KUKA KRL program: f1_Kuka_APT217T03S17.SRC

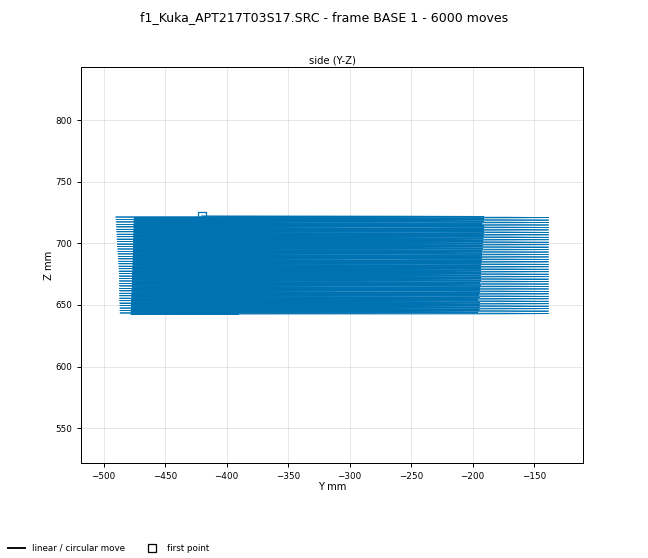
[picture p0: tool path of f1_Kuka_APT217T03S17.SRC in frame BASE 1, 6000 of 6001 moves have a stored position in this frame; points joined in program order, loops and branches not executed]
&ACCESS RVP
&REL 2
&PARAM TEMPLATE = C:\KRC\Roboter\Template\vorgabe
&PARAM EDITMASK = *
DEF f1_Kuka_APT217T03S17()


;FOLD INI;%{PE}%V3.2.0,%MKUKATPBASIS,%CINIT,%VCOMMON,%P
  ;FOLD BAS INI;%{E}%V3.2.0,%MKUKATPBASIS,%CINIT,%VINIT,%P
    GLOBAL INTERRUPT DECL 3 WHEN $STOPMESS==TRUE DO IR_STOPM ( )
    INTERRUPT ON 3
    BAS (#INITMOV,0 )
  ;ENDFOLD (BAS INI)
  ;FOLD USER INI;%{E}%V3.2.0,%MKUKATPUSER,%CINIT,%VINIT,%P
    ;Make your modifications here
  ;ENDFOLD (USER INI)
;ENDFOLD (INI)


;*** Make Null PTP Move
  PTP $pos_act

;*** Auto Load The Correct TOOL Data
  $tool=tool_data[3]

;*** Auto Load The Correct BASE Data
  $base=base_data[1]

  $ADVANCE = 5

;*** Restate Last Velocity
MMPM(30000.0)
SetRPM(6000)
LIN {X -0.045,Y -420.366,Z 722.490,A 0.000,B 0.000,C 90.000,E1 88.282} C_DIS
LIN {X -0.153,Y -409.375,Z 722.480,A 0.000,B 0.000,C 90.000,E1 86.388} C_DIS
LIN {X -0.011,Y -396.739,Z 722.467,A 0.000,B 0.000,C 90.000,E1 84.147} C_DIS
LIN {X -0.054,Y -382.651,Z 722.453,A 0.000,B 0.000,C 90.000,E1 81.602} C_DIS
LIN {X -0.034,Y -370.606,Z 722.440,A 0.000,B 0.000,C 90.000,E1 79.285} C_DIS
LIN {X -0.131,Y -357.568,Z 722.426,A 0.000,B 0.000,C 90.000,E1 76.645} C_DIS
LIN {X 0.016,Y -346.347,Z 722.412,A 0.000,B 0.000,C 90.000,E1 74.212} C_DIS
LIN {X -0.021,Y -335.329,Z 722.399,A 0.000,B 0.000,C 90.000,E1 71.764} C_DIS
LIN {X 0.156,Y -320.932,Z 722.380,A 0.000,B 0.000,C 90.000,E1 68.284} C_DIS
LIN {X 0.051,Y -311.481,Z 722.365,A 0.000,B 0.000,C 90.000,E1 65.741} C_DIS
LIN {X 0.067,Y -300.034,Z 722.345,A 0.000,B 0.000,C 90.000,E1 62.153} C_DIS
LIN {X -0.118,Y -290.423,Z 722.327,A 0.000,B 0.000,C 90.000,E1 58.869} C_DIS
LIN {X -0.001,Y -281.361,Z 722.308,A 0.000,B 0.000,C 90.000,E1 55.468} C_DIS
LIN {X -0.016,Y -276.153,Z 722.297,A 0.000,B 0.000,C 90.000,E1 53.417} C_DIS
LIN {X 0.036,Y -270.874,Z 722.285,A 0.000,B 0.000,C 90.000,E1 51.331} C_DIS
LIN {X 0.116,Y -265.448,Z 722.274,A 0.000,B 0.000,C 90.000,E1 49.218} C_DIS
LIN {X -0.099,Y -259.838,Z 722.262,A 0.000,B 0.000,C 90.000,E1 47.148} C_DIS
LIN {X -0.064,Y -254.168,Z 722.250,A 0.000,B 0.000,C 90.000,E1 45.000} C_DIS
LIN {X -0.132,Y -248.317,Z 722.238,A 0.000,B 0.000,C 90.000,E1 42.852} C_DIS
LIN {X 0.051,Y -242.351,Z 722.226,A 0.000,B 0.000,C 90.000,E1 40.620} C_DIS
LIN {X -0.106,Y -232.554,Z 722.205,A 0.000,B 0.000,C 90.000,E1 36.950} C_DIS
LIN {X -0.091,Y -223.507,Z 722.184,A 0.000,B 0.000,C 90.000,E1 33.166} C_DIS
LIN {X -0.050,Y -216.883,Z 722.167,A 0.000,B 0.000,C 90.000,E1 30.079} C_DIS
LIN {X -0.011,Y -211.033,Z 722.150,A 0.000,B 0.000,C 90.000,E1 26.950} C_DIS
LIN {X 0.066,Y -205.943,Z 722.132,A 0.000,B 0.000,C 90.000,E1 23.770} C_DIS
LIN {X -0.046,Y -201.601,Z 722.114,A 0.000,B 0.000,C 90.000,E1 20.610} C_DIS
LIN {X -0.008,Y -197.203,Z 722.092,A 0.000,B 0.000,C 90.000,E1 16.567} C_DIS
LIN {X 0.070,Y -193.392,Z 722.065,A 0.000,B 0.000,C 90.000,E1 11.658} C_DIS
LIN {X 0.073,Y -190.840,Z 722.033,A 0.000,B 0.000,C 90.000,E1 5.910} C_DIS
LIN {X -0.076,Y -191.951,Z 721.970,A 0.000,B 0.000,C 90.000,E1 354.609} C_DIS
LIN {X -0.101,Y -194.807,Z 721.943,A 0.000,B 0.000,C 90.000,E1 349.690} C_DIS
LIN {X -0.024,Y -198.321,Z 721.920,A 0.000,B 0.000,C 90.000,E1 345.589} C_DIS
LIN {X 0.030,Y -202.840,Z 721.897,A 0.000,B 0.000,C 90.000,E1 341.529} C_DIS
LIN {X -0.017,Y -208.249,Z 721.875,A 0.000,B 0.000,C 90.000,E1 337.539} C_DIS
LIN {X -0.036,Y -214.509,Z 721.853,A 0.000,B 0.000,C 90.000,E1 333.589} C_DIS
LIN {X 0.047,Y -221.349,Z 721.832,A 0.000,B 0.000,C 90.000,E1 329.665} C_DIS
LIN {X 0.069,Y -227.297,Z 721.814,A 0.000,B 0.000,C 90.000,E1 326.580} C_DIS
LIN {X 0.013,Y -235.274,Z 721.793,A 0.000,B 0.000,C 90.000,E1 322.798} C_DIS
LIN {X 0.048,Y -243.974,Z 721.773,A 0.000,B 0.000,C 90.000,E1 319.057} C_DIS
LIN {X -0.019,Y -253.622,Z 721.752,A 0.000,B 0.000,C 90.000,E1 315.405} C_DIS
LIN {X -0.120,Y -264.412,Z 721.732,A 0.000,B 0.000,C 90.000,E1 311.838} C_DIS
LIN {X -0.010,Y -276.297,Z 721.713,A 0.000,B 0.000,C 90.000,E1 308.302} C_DIS
LIN {X -0.150,Y -289.563,Z 721.694,A 0.000,B 0.000,C 90.000,E1 304.898} C_DIS
LIN {X -0.111,Y -304.342,Z 721.675,A 0.000,B 0.000,C 90.000,E1 301.544} C_DIS
LIN {X -0.142,Y -319.094,Z 721.659,A 0.000,B 0.000,C 90.000,E1 298.615} C_DIS
LIN {X 0.051,Y -337.144,Z 721.641,A 0.000,B 0.000,C 90.000,E1 295.412} C_DIS
LIN {X 0.060,Y -354.682,Z 721.626,A 0.000,B 0.000,C 90.000,E1 292.642} C_DIS
LIN {X -0.097,Y -375.452,Z 721.609,A 0.000,B 0.000,C 90.000,E1 289.685} C_DIS
LIN {X -0.149,Y -396.197,Z 721.595,A 0.000,B 0.000,C 90.000,E1 287.094} C_DIS
LIN {X 0.119,Y -410.310,Z 721.586,A 0.000,B 0.000,C 90.000,E1 285.371} C_DIS
LIN {X 0.155,Y -424.096,Z 721.576,A 0.000,B 0.000,C 90.000,E1 283.716} C_DIS
LIN {X -0.176,Y -435.418,Z 721.569,A 0.000,B 0.000,C 90.000,E1 282.411} C_DIS
LIN {X 0.197,Y -444.037,Z 721.563,A 0.000,B 0.000,C 90.000,E1 281.299} C_DIS
LIN {X -0.035,Y -454.322,Z 721.556,A 0.000,B 0.000,C 90.000,E1 280.018} C_DIS
LIN {X 0.089,Y -466.419,Z 721.547,A 0.000,B 0.000,C 90.000,E1 278.454} C_DIS
LIN {X -0.153,Y -473.979,Z 721.541,A 0.000,B 0.000,C 90.000,E1 277.466} C_DIS
LIN {X -0.243,Y -478.914,Z 721.537,A 0.000,B 0.000,C 90.000,E1 276.720} C_DIS
LIN {X -0.096,Y -481.792,Z 721.534,A 0.000,B 0.000,C 90.000,E1 276.201} C_DIS
LIN {X 0.070,Y -484.223,Z 721.532,A 0.000,B 0.000,C 90.000,E1 275.682} C_DIS
LIN {X -0.232,Y -486.263,Z 721.529,A 0.000,B 0.000,C 90.000,E1 275.220} C_DIS
LIN {X -0.045,Y -487.865,Z 721.526,A 0.000,B 0.000,C 90.000,E1 274.702} C_DIS
LIN {X 0.115,Y -489.063,Z 721.523,A 0.000,B 0.000,C 90.000,E1 274.188} C_DIS
LIN {X -0.166,Y -489.824,Z 721.521,A 0.000,B 0.000,C 90.000,E1 273.726} C_DIS
LIN {X 0.017,Y -490.215,Z 721.518,A 0.000,B 0.000,C 90.000,E1 273.212} C_DIS
LIN {X 0.233,Y -490.237,Z 721.515,A 0.000,B 0.000,C 90.000,E1 272.694} C_DIS
LIN {X -0.063,Y -489.908,Z 721.512,A 0.000,B 0.000,C 90.000,E1 272.236} C_DIS
LIN {X 0.148,Y -489.291,Z 721.510,A 0.000,B 0.000,C 90.000,E1 271.718} C_DIS
LIN {X -0.148,Y -488.268,Z 721.507,A 0.000,B 0.000,C 90.000,E1 271.260} C_DIS
LIN {X 0.041,Y -486.857,Z 721.504,A 0.000,B 0.000,C 90.000,E1 270.745} C_DIS
LIN {X 0.225,Y -484.965,Z 721.501,A 0.000,B 0.000,C 90.000,E1 270.229} C_DIS
LIN {X -0.083,Y -482.513,Z 721.499,A 0.000,B 0.000,C 90.000,E1 269.771} C_DIS
LIN {X 0.074,Y -479.349,Z 721.496,A 0.000,B 0.000,C 90.000,E1 269.255} C_DIS
LIN {X 0.212,Y -475.359,Z 721.493,A 0.000,B 0.000,C 90.000,E1 268.740} C_DIS
LIN {X -0.144,Y -470.353,Z 721.490,A 0.000,B 0.000,C 90.000,E1 268.282} C_DIS
LIN {X -0.225,Y -467.502,Z 721.489,A 0.000,B 0.000,C 90.000,E1 268.051} C_DIS
LIN {X 0.144,Y -464.309,Z 721.488,A 0.000,B 0.000,C 90.000,E1 267.764} C_DIS
LIN {X 0.057,Y -457.761,Z 721.485,A 0.000,B 0.000,C 90.000,E1 267.364} C_DIS
LIN {X 0.057,Y -454.413,Z 721.484,A 0.000,B 0.000,C 90.000,E1 267.192} C_DIS
LIN {X -0.086,Y -447.138,Z 721.483,A 0.000,B 0.000,C 90.000,E1 266.906} C_DIS
LIN {X -0.114,Y -439.506,Z 721.481,A 0.000,B 0.000,C 90.000,E1 266.674} C_DIS
LIN {X -0.117,Y -431.202,Z 721.480,A 0.000,B 0.000,C 90.000,E1 266.502} C_DIS
LIN {X -0.201,Y -425.998,Z 721.480,A 0.000,B 0.000,C 90.000,E1 266.445} C_DIS
LIN {X -0.115,Y -419.753,Z 721.480,A 0.000,B 0.000,C 90.000,E1 266.388} C_DIS
LIN {X -0.086,Y -180.939,Z 721.480,A 0.000,B 0.000,C 90.000,E1 266.388} C_DIS
LIN {X -0.079,Y -180.742,Z 721.470,A 0.000,B 0.000,C 90.000,E1 264.666} C_DIS
LIN {X 0.022,Y -178.834,Z 721.442,A 0.000,B 0.000,C 90.000,E1 259.567} C_DIS
LIN {X 0.056,Y -175.878,Z 721.414,A 0.000,B 0.000,C 90.000,E1 254.464} C_DIS
LIN {X -0.007,Y -174.538,Z 721.404,A 0.000,B 0.000,C 90.000,E1 252.779} C_DIS
LIN {X 0.086,Y -171.522,Z 721.380,A 0.000,B 0.000,C 90.000,E1 248.465} C_DIS
LIN {X 0.071,Y -167.748,Z 721.357,A 0.000,B 0.000,C 90.000,E1 244.152} C_DIS
LIN {X 0.010,Y -166.451,Z 721.347,A 0.000,B 0.000,C 90.000,E1 242.436} C_DIS
LIN {X 0.000,Y -163.167,Z 721.328,A 0.000,B 0.000,C 90.000,E1 238.948} C_DIS
LIN {X 0.049,Y -161.126,Z 721.313,A 0.000,B 0.000,C 90.000,E1 236.294} C_DIS
LIN {X -0.048,Y -157.149,Z 721.288,A 0.000,B 0.000,C 90.000,E1 231.904} C_DIS
LIN {X -0.025,Y -155.880,Z 721.278,A 0.000,B 0.000,C 90.000,E1 230.114} C_DIS
LIN {X -0.066,Y -152.131,Z 721.253,A 0.000,B 0.000,C 90.000,E1 225.648} C_DIS
LIN {X -0.046,Y -150.381,Z 721.238,A 0.000,B 0.000,C 90.000,E1 222.933} C_DIS
LIN {X -0.021,Y -147.113,Z 721.213,A 0.000,B 0.000,C 90.000,E1 218.382} C_DIS
LIN {X -0.030,Y -145.679,Z 721.198,A 0.000,B 0.000,C 90.000,E1 215.644} C_DIS
LIN {X -0.032,Y -143.061,Z 721.172,A 0.000,B 0.000,C 90.000,E1 211.052} C_DIS
LIN {X 0.025,Y -141.683,Z 721.152,A 0.000,B 0.000,C 90.000,E1 207.334} C_DIS
LIN {X 0.004,Y -139.458,Z 721.116,A 0.000,B 0.000,C 90.000,E1 200.844} C_DIS
LIN {X 0.055,Y -139.192,Z 721.105,A 0.000,B 0.000,C 90.000,E1 198.960} C_DIS
LIN {X -0.058,Y -138.324,Z 721.054,A 0.000,B 0.000,C 90.000,E1 189.670} C_DIS
LIN {X -0.054,Y -139.455,Z 721.007,A 0.000,B 0.000,C 90.000,E1 181.260} C_DIS
LIN {X 0.026,Y -141.003,Z 720.976,A 0.000,B 0.000,C 90.000,E1 175.641} C_DIS
LIN {X -0.024,Y -142.757,Z 720.955,A 0.000,B 0.000,C 90.000,E1 171.951} C_DIS
LIN {X -0.069,Y -145.160,Z 720.930,A 0.000,B 0.000,C 90.000,E1 167.353} C_DIS
LIN {X -0.077,Y -147.783,Z 720.909,A 0.000,B 0.000,C 90.000,E1 163.685} C_DIS
LIN {X 0.003,Y -150.462,Z 720.889,A 0.000,B 0.000,C 90.000,E1 160.007} C_DIS
LIN {X 0.077,Y -153.913,Z 720.869,A 0.000,B 0.000,C 90.000,E1 156.357} C_DIS
LIN {X 0.002,Y -157.323,Z 720.849,A 0.000,B 0.000,C 90.000,E1 152.794} C_DIS
LIN {X 0.086,Y -161.512,Z 720.829,A 0.000,B 0.000,C 90.000,E1 149.203} C_DIS
LIN {X -0.037,Y -165.711,Z 720.810,A 0.000,B 0.000,C 90.000,E1 145.722} C_DIS
LIN {X 0.088,Y -170.657,Z 720.790,A 0.000,B 0.000,C 90.000,E1 142.190} C_DIS
LIN {X 0.001,Y -175.533,Z 720.771,A 0.000,B 0.000,C 90.000,E1 138.771} C_DIS
LIN {X -0.006,Y -181.152,Z 720.752,A 0.000,B 0.000,C 90.000,E1 135.364} C_DIS
LIN {X -0.007,Y -186.606,Z 720.733,A 0.000,B 0.000,C 90.000,E1 132.000} C_DIS
LIN {X 0.028,Y -191.565,Z 720.718,A 0.000,B 0.000,C 90.000,E1 129.277} C_DIS
LIN {X 0.008,Y -290.263,Z 720.718,A 0.000,B 0.000,C 90.000,E1 129.277} C_DIS
LIN {X 0.150,Y -292.744,Z 720.718,A 0.000,B 0.000,C 90.000,E1 129.197} C_DIS
LIN {X -0.022,Y -297.486,Z 720.716,A 0.000,B 0.000,C 90.000,E1 128.955} C_DIS
LIN {X 0.033,Y -300.182,Z 720.715,A 0.000,B 0.000,C 90.000,E1 128.669} C_DIS
LIN {X 0.012,Y -303.878,Z 720.712,A 0.000,B 0.000,C 90.000,E1 128.096} C_DIS
LIN {X 0.204,Y -305.355,Z 720.710,A 0.000,B 0.000,C 90.000,E1 127.729} C_DIS
LIN {X -0.032,Y -306.516,Z 720.708,A 0.000,B 0.000,C 90.000,E1 127.443} C_DIS
LIN {X -0.049,Y -317.229,Z 720.688,A 0.000,B 0.000,C 90.000,E1 123.865} C_DIS
LIN {X -0.123,Y -327.331,Z 720.672,A 0.000,B 0.000,C 90.000,E1 121.003} C_DIS
LIN {X 0.034,Y -338.764,Z 720.656,A 0.000,B 0.000,C 90.000,E1 118.153} C_DIS
LIN {X -0.121,Y -351.632,Z 720.641,A 0.000,B 0.000,C 90.000,E1 115.412} C_DIS
LIN {X 0.208,Y -364.364,Z 720.628,A 0.000,B 0.000,C 90.000,E1 112.950} C_DIS
LIN {X 0.099,Y -378.411,Z 720.615,A 0.000,B 0.000,C 90.000,E1 110.610} C_DIS
LIN {X 0.079,Y -393.872,Z 720.602,A 0.000,B 0.000,C 90.000,E1 108.308} C_DIS
LIN {X -0.062,Y -410.861,Z 720.589,A 0.000,B 0.000,C 90.000,E1 106.079} C_DIS
LIN {X -0.026,Y -429.500,Z 720.577,A 0.000,B 0.000,C 90.000,E1 103.883} C_DIS
LIN {X 0.195,Y -449.465,Z 720.566,A 0.000,B 0.000,C 90.000,E1 101.771} C_DIS
LIN {X -0.208,Y -467.386,Z 720.556,A 0.000,B 0.000,C 90.000,E1 100.141} C_DIS
LIN {X -0.172,Y -469.669,Z 720.555,A 0.000,B 0.000,C 90.000,E1 99.905} C_DIS
LIN {X 0.177,Y -471.507,Z 720.554,A 0.000,B 0.000,C 90.000,E1 99.613} C_DIS
LIN {X 0.061,Y -472.893,Z 720.552,A 0.000,B 0.000,C 90.000,E1 99.378} C_DIS
LIN {X 0.168,Y -474.683,Z 720.549,A 0.000,B 0.000,C 90.000,E1 98.859} C_DIS
LIN {X -0.185,Y -475.386,Z 720.547,A 0.000,B 0.000,C 90.000,E1 98.398} C_DIS
LIN {X 0.010,Y -475.120,Z 720.544,A 0.000,B 0.000,C 90.000,E1 97.871} C_DIS
LIN {X 0.142,Y -473.850,Z 720.541,A 0.000,B 0.000,C 90.000,E1 97.352} C_DIS
LIN {X -0.056,Y -472.778,Z 720.540,A 0.000,B 0.000,C 90.000,E1 97.125} C_DIS
LIN {X 0.071,Y -469.662,Z 720.537,A 0.000,B 0.000,C 90.000,E1 96.606} C_DIS
LIN {X -0.074,Y -453.400,Z 720.523,A 0.000,B 0.000,C 90.000,E1 94.073} C_DIS
LIN {X 0.011,Y -440.049,Z 720.510,A 0.000,B 0.000,C 90.000,E1 91.718} C_DIS
LIN {X 0.130,Y -431.084,Z 720.501,A 0.000,B 0.000,C 90.000,E1 90.115} C_DIS
LIN {X -0.215,Y -420.296,Z 720.490,A 0.000,B 0.000,C 90.000,E1 88.282} C_DIS
LIN {X 0.088,Y -409.303,Z 720.480,A 0.000,B 0.000,C 90.000,E1 86.331} C_DIS
LIN {X -0.174,Y -396.689,Z 720.467,A 0.000,B 0.000,C 90.000,E1 84.147} C_DIS
LIN {X 0.200,Y -381.112,Z 720.452,A 0.000,B 0.000,C 90.000,E1 81.254} C_DIS
LIN {X -0.189,Y -369.132,Z 720.439,A 0.000,B 0.000,C 90.000,E1 78.993} C_DIS
LIN {X 0.022,Y -356.168,Z 720.424,A 0.000,B 0.000,C 90.000,E1 76.297} C_DIS
LIN {X 0.123,Y -344.996,Z 720.410,A 0.000,B 0.000,C 90.000,E1 73.866} C_DIS
LIN {X 0.131,Y -332.686,Z 720.395,A 0.000,B 0.000,C 90.000,E1 71.094} C_DIS
LIN {X -0.081,Y -318.566,Z 720.376,A 0.000,B 0.000,C 90.000,E1 67.667} C_DIS
LIN {X -0.023,Y -310.507,Z 720.363,A 0.000,B 0.000,C 90.000,E1 65.409} C_DIS
LIN {X -0.049,Y -300.214,Z 720.345,A 0.000,B 0.000,C 90.000,E1 62.153} C_DIS
LIN {X 0.024,Y -290.640,Z 720.327,A 0.000,B 0.000,C 90.000,E1 58.820} C_DIS
LIN {X -0.097,Y -281.608,Z 720.308,A 0.000,B 0.000,C 90.000,E1 55.468} C_DIS
LIN {X -0.106,Y -276.420,Z 720.297,A 0.000,B 0.000,C 90.000,E1 53.417} C_DIS
LIN {X -0.048,Y -271.151,Z 720.285,A 0.000,B 0.000,C 90.000,E1 51.331} C_DIS
LIN {X 0.040,Y -265.742,Z 720.273,A 0.000,B 0.000,C 90.000,E1 49.218} C_DIS
LIN {X 0.022,Y -260.146,Z 720.262,A 0.000,B 0.000,C 90.000,E1 47.106} C_DIS
LIN {X -0.125,Y -254.445,Z 720.250,A 0.000,B 0.000,C 90.000,E1 45.000} C_DIS
LIN {X -0.018,Y -248.610,Z 720.238,A 0.000,B 0.000,C 90.000,E1 42.813} C_DIS
LIN {X 0.002,Y -242.609,Z 720.226,A 0.000,B 0.000,C 90.000,E1 40.620} C_DIS
LIN {X -0.005,Y -232.771,Z 720.205,A 0.000,B 0.000,C 90.000,E1 36.916} C_DIS
LIN {X -0.122,Y -223.698,Z 720.184,A 0.000,B 0.000,C 90.000,E1 33.166} C_DIS
LIN {X 0.033,Y -217.037,Z 720.167,A 0.000,B 0.000,C 90.000,E1 30.050} C_DIS
LIN {X -0.032,Y -211.188,Z 720.150,A 0.000,B 0.000,C 90.000,E1 26.950} C_DIS
LIN {X 0.049,Y -206.089,Z 720.132,A 0.000,B 0.000,C 90.000,E1 23.770} C_DIS
LIN {X -0.060,Y -201.735,Z 720.114,A 0.000,B 0.000,C 90.000,E1 20.610} C_DIS
LIN {X 0.040,Y -197.327,Z 720.092,A 0.000,B 0.000,C 90.000,E1 16.551} C_DIS
LIN {X 0.054,Y -194.024,Z 720.069,A 0.000,B 0.000,C 90.000,E1 12.479} C_DIS
LIN {X -0.073,Y -191.194,Z 720.038,A 0.000,B 0.000,C 90.000,E1 6.777} C_DIS
LIN {X 0.076,Y -192.439,Z 719.965,A 0.000,B 0.000,C 90.000,E1 353.742} C_DIS
LIN {X -0.084,Y -195.552,Z 719.938,A 0.000,B 0.000,C 90.000,E1 348.870} C_DIS
LIN {X 0.067,Y -199.250,Z 719.915,A 0.000,B 0.000,C 90.000,E1 344.755} C_DIS
LIN {X 0.023,Y -203.948,Z 719.893,A 0.000,B 0.000,C 90.000,E1 340.732} C_DIS
LIN {X 0.013,Y -209.531,Z 719.871,A 0.000,B 0.000,C 90.000,E1 336.741} C_DIS
LIN {X 0.026,Y -215.881,Z 719.849,A 0.000,B 0.000,C 90.000,E1 332.794} C_DIS
LIN {X -0.028,Y -222.851,Z 719.827,A 0.000,B 0.000,C 90.000,E1 328.918} C_DIS
LIN {X -0.092,Y -230.456,Z 719.806,A 0.000,B 0.000,C 90.000,E1 325.102} C_DIS
LIN {X -0.097,Y -238.696,Z 719.785,A 0.000,B 0.000,C 90.000,E1 321.331} C_DIS
LIN {X 0.023,Y -247.740,Z 719.764,A 0.000,B 0.000,C 90.000,E1 317.595} C_DIS
LIN {X -0.121,Y -256.774,Z 719.746,A 0.000,B 0.000,C 90.000,E1 314.352} C_DIS
LIN {X -0.107,Y -267.869,Z 719.726,A 0.000,B 0.000,C 90.000,E1 310.782} C_DIS
LIN {X 0.056,Y -278.884,Z 719.709,A 0.000,B 0.000,C 90.000,E1 307.604} C_DIS
LIN {X 0.010,Y -292.442,Z 719.690,A 0.000,B 0.000,C 90.000,E1 304.199} C_DIS
LIN {X -0.039,Y -305.944,Z 719.673,A 0.000,B 0.000,C 90.000,E1 301.209} C_DIS
LIN {X -0.093,Y -319.107,Z 719.659,A 0.000,B 0.000,C 90.000,E1 298.615} C_DIS
LIN {X 0.103,Y -337.113,Z 719.641,A 0.000,B 0.000,C 90.000,E1 295.412} C_DIS
LIN {X 0.113,Y -354.597,Z 719.626,A 0.000,B 0.000,C 90.000,E1 292.642} C_DIS
LIN {X -0.043,Y -375.337,Z 719.609,A 0.000,B 0.000,C 90.000,E1 289.685} C_DIS
LIN {X -0.096,Y -396.044,Z 719.595,A 0.000,B 0.000,C 90.000,E1 287.094} C_DIS
LIN {X 0.171,Y -410.128,Z 719.586,A 0.000,B 0.000,C 90.000,E1 285.371} C_DIS
LIN {X -0.206,Y -423.888,Z 719.576,A 0.000,B 0.000,C 90.000,E1 283.772} C_DIS
LIN {X -0.127,Y -435.207,Z 719.569,A 0.000,B 0.000,C 90.000,E1 282.411} C_DIS
LIN {X 0.244,Y -443.843,Z 719.563,A 0.000,B 0.000,C 90.000,E1 281.299} C_DIS
LIN {X 0.010,Y -454.095,Z 719.556,A 0.000,B 0.000,C 90.000,E1 280.018} C_DIS
LIN {X 0.131,Y -466.190,Z 719.547,A 0.000,B 0.000,C 90.000,E1 278.454} C_DIS
LIN {X -0.113,Y -473.775,Z 719.541,A 0.000,B 0.000,C 90.000,E1 277.466} C_DIS
LIN {X -0.204,Y -478.702,Z 719.537,A 0.000,B 0.000,C 90.000,E1 276.720} C_DIS
LIN {X -0.058,Y -481.588,Z 719.534,A 0.000,B 0.000,C 90.000,E1 276.201} C_DIS
LIN {X 0.107,Y -484.034,Z 719.532,A 0.000,B 0.000,C 90.000,E1 275.682} C_DIS
LIN {X -0.196,Y -486.084,Z 719.529,A 0.000,B 0.000,C 90.000,E1 275.220} C_DIS
LIN {X -0.004,Y -487.694,Z 719.526,A 0.000,B 0.000,C 90.000,E1 274.702} C_DIS
LIN {X 0.156,Y -488.877,Z 719.523,A 0.000,B 0.000,C 90.000,E1 274.188} C_DIS
LIN {X -0.126,Y -489.635,Z 719.521,A 0.000,B 0.000,C 90.000,E1 273.726} C_DIS
LIN {X 0.056,Y -489.999,Z 719.518,A 0.000,B 0.000,C 90.000,E1 273.212} C_DIS
LIN {X -0.219,Y -490.051,Z 719.515,A 0.000,B 0.000,C 90.000,E1 272.751} C_DIS
LIN {X -0.027,Y -489.687,Z 719.512,A 0.000,B 0.000,C 90.000,E1 272.236} C_DIS
LIN {X 0.183,Y -489.091,Z 719.510,A 0.000,B 0.000,C 90.000,E1 271.718} C_DIS
LIN {X -0.115,Y -488.083,Z 719.507,A 0.000,B 0.000,C 90.000,E1 271.260} C_DIS
LIN {X 0.074,Y -486.677,Z 719.504,A 0.000,B 0.000,C 90.000,E1 270.745} C_DIS
LIN {X -0.228,Y -484.823,Z 719.501,A 0.000,B 0.000,C 90.000,E1 270.286} C_DIS
LIN {X -0.052,Y -482.380,Z 719.499,A 0.000,B 0.000,C 90.000,E1 269.771} C_DIS
LIN {X 0.103,Y -479.214,Z 719.496,A 0.000,B 0.000,C 90.000,E1 269.255} C_DIS
LIN {X -0.235,Y -475.261,Z 719.493,A 0.000,B 0.000,C 90.000,E1 268.797} C_DIS
LIN {X -0.116,Y -470.303,Z 719.490,A 0.000,B 0.000,C 90.000,E1 268.282} C_DIS
LIN {X -0.200,Y -467.490,Z 719.489,A 0.000,B 0.000,C 90.000,E1 268.051} C_DIS
LIN {X 0.167,Y -464.322,Z 719.488,A 0.000,B 0.000,C 90.000,E1 267.764} C_DIS
LIN {X -0.119,Y -461.259,Z 719.487,A 0.000,B 0.000,C 90.000,E1 267.593} C_DIS
LIN {X 0.057,Y -457.778,Z 719.485,A 0.000,B 0.000,C 90.000,E1 267.364} C_DIS
LIN {X 0.053,Y -450.582,Z 719.483,A 0.000,B 0.000,C 90.000,E1 267.020} C_DIS
LIN {X 0.210,Y -443.185,Z 719.482,A 0.000,B 0.000,C 90.000,E1 266.731} C_DIS
LIN {X -0.066,Y -435.015,Z 719.481,A 0.000,B 0.000,C 90.000,E1 266.560} C_DIS
LIN {X 0.107,Y -425.230,Z 719.480,A 0.000,B 0.000,C 90.000,E1 266.388} C_DIS
LIN {X 0.192,Y -417.389,Z 719.480,A 0.000,B 0.000,C 90.000,E1 266.331} C_DIS
LIN {X 0.048,Y -180.938,Z 719.480,A 0.000,B 0.000,C 90.000,E1 266.331} C_DIS
LIN {X 0.055,Y -180.736,Z 719.470,A 0.000,B 0.000,C 90.000,E1 264.609} C_DIS
LIN {X -0.024,Y -178.826,Z 719.442,A 0.000,B 0.000,C 90.000,E1 259.567} C_DIS
LIN {X 0.058,Y -175.870,Z 719.414,A 0.000,B 0.000,C 90.000,E1 254.448} C_DIS
LIN {X 0.052,Y -173.843,Z 719.399,A 0.000,B 0.000,C 90.000,E1 251.891} C_DIS
LIN {X 0.041,Y -171.511,Z 719.380,A 0.000,B 0.000,C 90.000,E1 248.465} C_DIS
LIN {X 0.028,Y -167.738,Z 719.356,A 0.000,B 0.000,C 90.000,E1 244.152} C_DIS
LIN {X 0.044,Y -166.437,Z 719.347,A 0.000,B 0.000,C 90.000,E1 242.410} C_DIS
LIN {X -0.043,Y -163.155,Z 719.327,A 0.000,B 0.000,C 90.000,E1 238.948} C_DIS
LIN {X 0.007,Y -161.112,Z 719.313,A 0.000,B 0.000,C 90.000,E1 236.294} C_DIS
LIN {X -0.010,Y -157.837,Z 719.293,A 0.000,B 0.000,C 90.000,E1 232.763} C_DIS
LIN {X 0.053,Y -155.870,Z 719.278,A 0.000,B 0.000,C 90.000,E1 230.070} C_DIS
LIN {X 0.001,Y -152.120,Z 719.253,A 0.000,B 0.000,C 90.000,E1 225.607} C_DIS
LIN {X 0.016,Y -150.370,Z 719.238,A 0.000,B 0.000,C 90.000,E1 222.894} C_DIS
LIN {X -0.062,Y -147.104,Z 719.213,A 0.000,B 0.000,C 90.000,E1 218.382} C_DIS
LIN {X 0.048,Y -145.673,Z 719.198,A 0.000,B 0.000,C 90.000,E1 215.598} C_DIS
LIN {X 0.051,Y -143.054,Z 719.172,A 0.000,B 0.000,C 90.000,E1 211.003} C_DIS
LIN {X -0.013,Y -141.677,Z 719.152,A 0.000,B 0.000,C 90.000,E1 207.334} C_DIS
LIN {X -0.035,Y -139.455,Z 719.116,A 0.000,B 0.000,C 90.000,E1 200.844} C_DIS
LIN {X 0.016,Y -139.189,Z 719.105,A 0.000,B 0.000,C 90.000,E1 198.960} C_DIS
LIN {X 0.039,Y -138.323,Z 719.053,A 0.000,B 0.000,C 90.000,E1 189.613} C_DIS
LIN {X 0.046,Y -139.458,Z 719.007,A 0.000,B 0.000,C 90.000,E1 181.203} C_DIS
LIN {X -0.013,Y -141.009,Z 718.976,A 0.000,B 0.000,C 90.000,E1 175.641} C_DIS
LIN {X -0.064,Y -142.763,Z 718.955,A 0.000,B 0.000,C 90.000,E1 171.951} C_DIS
LIN {X 0.033,Y -145.170,Z 718.930,A 0.000,B 0.000,C 90.000,E1 167.297} C_DIS
LIN {X 0.025,Y -147.792,Z 718.909,A 0.000,B 0.000,C 90.000,E1 163.630} C_DIS
LIN {X -0.039,Y -150.475,Z 718.889,A 0.000,B 0.000,C 90.000,E1 160.007} C_DIS
LIN {X 0.036,Y -153.929,Z 718.869,A 0.000,B 0.000,C 90.000,E1 156.357} C_DIS
LIN {X -0.041,Y -157.339,Z 718.849,A 0.000,B 0.000,C 90.000,E1 152.794} C_DIS
LIN {X 0.043,Y -161.532,Z 718.829,A 0.000,B 0.000,C 90.000,E1 149.203} C_DIS
LIN {X 0.056,Y -165.730,Z 718.809,A 0.000,B 0.000,C 90.000,E1 145.674} C_DIS
LIN {X 0.044,Y -170.680,Z 718.790,A 0.000,B 0.000,C 90.000,E1 142.190} C_DIS
LIN {X -0.043,Y -175.555,Z 718.771,A 0.000,B 0.000,C 90.000,E1 138.771} C_DIS
LIN {X 0.076,Y -181.173,Z 718.752,A 0.000,B 0.000,C 90.000,E1 135.324} C_DIS
LIN {X -0.054,Y -186.631,Z 718.733,A 0.000,B 0.000,C 90.000,E1 132.000} C_DIS
LIN {X 0.072,Y -191.544,Z 718.718,A 0.000,B 0.000,C 90.000,E1 129.277} C_DIS
LIN {X 0.058,Y -290.577,Z 718.718,A 0.000,B 0.000,C 90.000,E1 129.277} C_DIS
LIN {X 0.043,Y -295.194,Z 718.717,A 0.000,B 0.000,C 90.000,E1 129.116} C_DIS
LIN {X -0.109,Y -297.362,Z 718.716,A 0.000,B 0.000,C 90.000,E1 128.991} C_DIS
LIN {X -0.040,Y -300.349,Z 718.715,A 0.000,B 0.000,C 90.000,E1 128.669} C_DIS
LIN {X -0.092,Y -303.985,Z 718.712,A 0.000,B 0.000,C 90.000,E1 128.096} C_DIS
LIN {X 0.101,Y -305.426,Z 718.710,A 0.000,B 0.000,C 90.000,E1 127.729} C_DIS
LIN {X -0.135,Y -306.559,Z 718.708,A 0.000,B 0.000,C 90.000,E1 127.443} C_DIS
LIN {X 0.023,Y -317.270,Z 718.688,A 0.000,B 0.000,C 90.000,E1 123.833} C_DIS
LIN {X 0.219,Y -327.381,Z 718.672,A 0.000,B 0.000,C 90.000,E1 120.924} C_DIS
LIN {X -0.075,Y -338.822,Z 718.656,A 0.000,B 0.000,C 90.000,E1 118.153} C_DIS
LIN {X -0.082,Y -351.700,Z 718.641,A 0.000,B 0.000,C 90.000,E1 115.387} C_DIS
LIN {X 0.093,Y -364.442,Z 718.628,A 0.000,B 0.000,C 90.000,E1 112.950} C_DIS
LIN {X -0.018,Y -378.497,Z 718.615,A 0.000,B 0.000,C 90.000,E1 110.610} C_DIS
LIN {X -0.040,Y -393.970,Z 718.602,A 0.000,B 0.000,C 90.000,E1 108.308} C_DIS
LIN {X -0.184,Y -410.970,Z 718.589,A 0.000,B 0.000,C 90.000,E1 106.079} C_DIS
LIN {X -0.151,Y -429.623,Z 718.577,A 0.000,B 0.000,C 90.000,E1 103.883} C_DIS
LIN {X 0.074,Y -449.592,Z 718.565,A 0.000,B 0.000,C 90.000,E1 101.771} C_DIS
LIN {X 0.218,Y -467.517,Z 718.556,A 0.000,B 0.000,C 90.000,E1 100.074} C_DIS
LIN {X 0.175,Y -469.775,Z 718.555,A 0.000,B 0.000,C 90.000,E1 99.849} C_DIS
LIN {X 0.047,Y -471.604,Z 718.553,A 0.000,B 0.000,C 90.000,E1 99.613} C_DIS
LIN {X -0.082,Y -472.982,Z 718.552,A 0.000,B 0.000,C 90.000,E1 99.378} C_DIS
LIN {X 0.025,Y -474.745,Z 718.549,A 0.000,B 0.000,C 90.000,E1 98.859} C_DIS
LIN {X 0.144,Y -475.426,Z 718.546,A 0.000,B 0.000,C 90.000,E1 98.341} C_DIS
LIN {X -0.130,Y -475.137,Z 718.544,A 0.000,B 0.000,C 90.000,E1 97.871} C_DIS
LIN {X 0.002,Y -473.843,Z 718.541,A 0.000,B 0.000,C 90.000,E1 97.352} C_DIS
LIN {X -0.197,Y -472.755,Z 718.539,A 0.000,B 0.000,C 90.000,E1 97.125} C_DIS
LIN {X -0.070,Y -469.622,Z 718.537,A 0.000,B 0.000,C 90.000,E1 96.606} C_DIS
LIN {X -0.178,Y -453.354,Z 718.522,A 0.000,B 0.000,C 90.000,E1 94.069} C_DIS
LIN {X 0.053,Y -438.543,Z 718.508,A 0.000,B 0.000,C 90.000,E1 91.432} C_DIS
LIN {X 0.145,Y -429.518,Z 718.499,A 0.000,B 0.000,C 90.000,E1 89.828} C_DIS
LIN {X 0.076,Y -420.258,Z 718.490,A 0.000,B 0.000,C 90.000,E1 88.224} C_DIS
LIN {X -0.038,Y -409.262,Z 718.480,A 0.000,B 0.000,C 90.000,E1 86.331} C_DIS
LIN {X 0.097,Y -396.675,Z 718.467,A 0.000,B 0.000,C 90.000,E1 84.090} C_DIS
LIN {X 0.082,Y -381.129,Z 718.451,A 0.000,B 0.000,C 90.000,E1 81.254} C_DIS
LIN {X 0.122,Y -367.680,Z 718.437,A 0.000,B 0.000,C 90.000,E1 78.634} C_DIS
LIN {X -0.003,Y -356.225,Z 718.424,A 0.000,B 0.000,C 90.000,E1 76.284} C_DIS
LIN {X 0.018,Y -345.062,Z 718.410,A 0.000,B 0.000,C 90.000,E1 73.866} C_DIS
LIN {X 0.045,Y -334.107,Z 718.397,A 0.000,B 0.000,C 90.000,E1 71.402} C_DIS
LIN {X -0.172,Y -318.686,Z 718.376,A 0.000,B 0.000,C 90.000,E1 67.667} C_DIS
LIN {X 0.130,Y -308.517,Z 718.360,A 0.000,B 0.000,C 90.000,E1 64.717} C_DIS
LIN {X 0.039,Y -298.449,Z 718.341,A 0.000,B 0.000,C 90.000,E1 61.463} C_DIS
LIN {X 0.105,Y -290.874,Z 718.327,A 0.000,B 0.000,C 90.000,E1 58.791} C_DIS
LIN {X 0.002,Y -281.877,Z 718.308,A 0.000,B 0.000,C 90.000,E1 55.435} C_DIS
LIN {X -0.160,Y -276.704,Z 718.297,A 0.000,B 0.000,C 90.000,E1 53.417} C_DIS
LIN {X -0.096,Y -271.447,Z 718.285,A 0.000,B 0.000,C 90.000,E1 51.331} C_DIS
LIN {X -0.002,Y -266.063,Z 718.273,A 0.000,B 0.000,C 90.000,E1 49.218} C_DIS
LIN {X -0.013,Y -260.466,Z 718.262,A 0.000,B 0.000,C 90.000,E1 47.106} C_DIS
LIN {X 0.026,Y -254.737,Z 718.250,A 0.000,B 0.000,C 90.000,E1 44.960} C_DIS
LIN {X 0.142,Y -248.906,Z 718.238,A 0.000,B 0.000,C 90.000,E1 42.771} C_DIS
LIN {X -0.014,Y -242.890,Z 718.226,A 0.000,B 0.000,C 90.000,E1 40.620} C_DIS
LIN {X -0.012,Y -233.007,Z 718.205,A 0.000,B 0.000,C 90.000,E1 36.916} C_DIS
LIN {X -0.123,Y -223.906,Z 718.184,A 0.000,B 0.000,C 90.000,E1 33.166} C_DIS
LIN {X -0.071,Y -217.206,Z 718.167,A 0.000,B 0.000,C 90.000,E1 30.079} C_DIS
LIN {X -0.023,Y -211.340,Z 718.150,A 0.000,B 0.000,C 90.000,E1 26.950} C_DIS
LIN {X 0.062,Y -206.242,Z 718.132,A 0.000,B 0.000,C 90.000,E1 23.770} C_DIS
LIN {X -0.043,Y -201.891,Z 718.114,A 0.000,B 0.000,C 90.000,E1 20.610} C_DIS
LIN {X 0.004,Y -197.459,Z 718.092,A 0.000,B 0.000,C 90.000,E1 16.567} C_DIS
LIN {X 0.077,Y -194.146,Z 718.069,A 0.000,B 0.000,C 90.000,E1 12.479} C_DIS
LIN {X -0.044,Y -191.333,Z 718.038,A 0.000,B 0.000,C 90.000,E1 6.777} C_DIS
LIN {X 0.082,Y -192.564,Z 717.965,A 0.000,B 0.000,C 90.000,E1 353.742} C_DIS
LIN {X -0.074,Y -195.669,Z 717.938,A 0.000,B 0.000,C 90.000,E1 348.870} C_DIS
LIN {X 0.081,Y -199.359,Z 717.915,A 0.000,B 0.000,C 90.000,E1 344.755} C_DIS
LIN {X 0.041,Y -204.045,Z 717.893,A 0.000,B 0.000,C 90.000,E1 340.732} C_DIS
LIN {X 0.034,Y -209.622,Z 717.871,A 0.000,B 0.000,C 90.000,E1 336.741} C_DIS
LIN {X 0.050,Y -215.944,Z 717.849,A 0.000,B 0.000,C 90.000,E1 332.794} C_DIS
LIN {X -0.001,Y -222.898,Z 717.827,A 0.000,B 0.000,C 90.000,E1 328.918} C_DIS
LIN {X -0.062,Y -230.501,Z 717.806,A 0.000,B 0.000,C 90.000,E1 325.102} C_DIS
LIN {X -0.065,Y -238.721,Z 717.785,A 0.000,B 0.000,C 90.000,E1 321.331} C_DIS
LIN {X -0.110,Y -247.739,Z 717.764,A 0.000,B 0.000,C 90.000,E1 317.634} C_DIS
LIN {X -0.085,Y -256.799,Z 717.746,A 0.000,B 0.000,C 90.000,E1 314.352} C_DIS
LIN {X -0.133,Y -266.735,Z 717.728,A 0.000,B 0.000,C 90.000,E1 311.148} C_DIS
LIN {X -0.003,Y -277.625,Z 717.711,A 0.000,B 0.000,C 90.000,E1 307.971} C_DIS
LIN {X 0.076,Y -291.056,Z 717.692,A 0.000,B 0.000,C 90.000,E1 304.532} C_DIS
LIN {X 0.007,Y -305.979,Z 717.673,A 0.000,B 0.000,C 90.000,E1 301.209} C_DIS
LIN {X 0.022,Y -320.853,Z 717.657,A 0.000,B 0.000,C 90.000,E1 298.281} C_DIS
LIN {X -0.176,Y -338.971,Z 717.640,A 0.000,B 0.000,C 90.000,E1 295.155} C_DIS
LIN {X -0.124,Y -356.543,Z 717.624,A 0.000,B 0.000,C 90.000,E1 292.386} C_DIS
LIN {X 0.010,Y -375.222,Z 717.609,A 0.000,B 0.000,C 90.000,E1 289.685} C_DIS
LIN {X -0.043,Y -395.893,Z 717.595,A 0.000,B 0.000,C 90.000,E1 287.094} C_DIS
LIN {X -0.164,Y -409.939,Z 717.586,A 0.000,B 0.000,C 90.000,E1 285.426} C_DIS
LIN {X 0.118,Y -421.384,Z 717.578,A 0.000,B 0.000,C 90.000,E1 284.008} C_DIS
LIN {X -0.070,Y -434.987,Z 717.569,A 0.000,B 0.000,C 90.000,E1 282.411} C_DIS
LIN {X -0.222,Y -443.629,Z 717.563,A 0.000,B 0.000,C 90.000,E1 281.366} C_DIS
LIN {X 0.064,Y -453.861,Z 717.556,A 0.000,B 0.000,C 90.000,E1 280.018} C_DIS
LIN {X 0.183,Y -465.944,Z 717.547,A 0.000,B 0.000,C 90.000,E1 278.454} C_DIS
LIN {X -0.064,Y -473.553,Z 717.541,A 0.000,B 0.000,C 90.000,E1 277.466} C_DIS
LIN {X -0.156,Y -478.537,Z 717.537,A 0.000,B 0.000,C 90.000,E1 276.720} C_DIS
LIN {X -0.145,Y -482.702,Z 717.533,A 0.000,B 0.000,C 90.000,E1 275.967} C_DIS
LIN {X -0.151,Y -485.888,Z 717.529,A 0.000,B 0.000,C 90.000,E1 275.220} C_DIS
LIN {X 0.034,Y -487.527,Z 717.526,A 0.000,B 0.000,C 90.000,E1 274.702} C_DIS
LIN {X 0.193,Y -488.684,Z 717.523,A 0.000,B 0.000,C 90.000,E1 274.188} C_DIS
LIN {X -0.090,Y -489.457,Z 717.521,A 0.000,B 0.000,C 90.000,E1 273.726} C_DIS
LIN {X 0.091,Y -489.829,Z 717.518,A 0.000,B 0.000,C 90.000,E1 273.212} C_DIS
LIN {X -0.185,Y -489.848,Z 717.515,A 0.000,B 0.000,C 90.000,E1 272.751} C_DIS
LIN {X 0.006,Y -489.542,Z 717.512,A 0.000,B 0.000,C 90.000,E1 272.236} C_DIS
LIN {X 0.215,Y -488.903,Z 717.510,A 0.000,B 0.000,C 90.000,E1 271.718} C_DIS
LIN {X -0.084,Y -487.934,Z 717.507,A 0.000,B 0.000,C 90.000,E1 271.260} C_DIS
LIN {X 0.103,Y -486.554,Z 717.504,A 0.000,B 0.000,C 90.000,E1 270.745} C_DIS
LIN {X -0.199,Y -484.686,Z 717.501,A 0.000,B 0.000,C 90.000,E1 270.286} C_DIS
LIN {X -0.025,Y -482.243,Z 717.499,A 0.000,B 0.000,C 90.000,E1 269.771} C_DIS
LIN {X 0.131,Y -479.103,Z 717.496,A 0.000,B 0.000,C 90.000,E1 269.255} C_DIS
LIN {X -0.208,Y -475.187,Z 717.493,A 0.000,B 0.000,C 90.000,E1 268.797} C_DIS
LIN {X -0.091,Y -470.280,Z 717.490,A 0.000,B 0.000,C 90.000,E1 268.282} C_DIS
LIN {X -0.193,Y -467.475,Z 717.489,A 0.000,B 0.000,C 90.000,E1 268.051} C_DIS
LIN {X 0.155,Y -464.300,Z 717.488,A 0.000,B 0.000,C 90.000,E1 267.764} C_DIS
LIN {X -0.139,Y -461.215,Z 717.487,A 0.000,B 0.000,C 90.000,E1 267.593} C_DIS
LIN {X 0.042,Y -454.391,Z 717.484,A 0.000,B 0.000,C 90.000,E1 267.192} C_DIS
LIN {X -0.124,Y -447.191,Z 717.483,A 0.000,B 0.000,C 90.000,E1 266.906} C_DIS
LIN {X -0.204,Y -439.353,Z 717.481,A 0.000,B 0.000,C 90.000,E1 266.674} C_DIS
LIN {X 0.173,Y -430.772,Z 717.480,A 0.000,B 0.000,C 90.000,E1 266.445} C_DIS
LIN {X -0.123,Y -422.610,Z 717.480,A 0.000,B 0.000,C 90.000,E1 266.388} C_DIS
LIN {X 0.125,Y -416.121,Z 717.480,A 0.000,B 0.000,C 90.000,E1 266.331} C_DIS
LIN {X 0.036,Y -180.938,Z 717.480,A 0.000,B 0.000,C 90.000,E1 266.331} C_DIS
LIN {X 0.023,Y -180.731,Z 717.470,A 0.000,B 0.000,C 90.000,E1 264.609} C_DIS
LIN {X -0.056,Y -178.821,Z 717.442,A 0.000,B 0.000,C 90.000,E1 259.567} C_DIS
LIN {X 0.026,Y -175.866,Z 717.414,A 0.000,B 0.000,C 90.000,E1 254.448} C_DIS
LIN {X 0.020,Y -173.834,Z 717.399,A 0.000,B 0.000,C 90.000,E1 251.891} C_DIS
LIN {X 0.010,Y -171.502,Z 717.380,A 0.000,B 0.000,C 90.000,E1 248.465} C_DIS
LIN {X -0.004,Y -167.730,Z 717.356,A 0.000,B 0.000,C 90.000,E1 244.152} C_DIS
LIN {X 0.013,Y -166.426,Z 717.347,A 0.000,B 0.000,C 90.000,E1 242.410} C_DIS
LIN {X 0.010,Y -163.146,Z 717.327,A 0.000,B 0.000,C 90.000,E1 238.918} C_DIS
LIN {X -0.024,Y -161.101,Z 717.313,A 0.000,B 0.000,C 90.000,E1 236.294} C_DIS
LIN {X -0.041,Y -157.829,Z 717.293,A 0.000,B 0.000,C 90.000,E1 232.763} C_DIS
LIN {X 0.023,Y -155.862,Z 717.278,A 0.000,B 0.000,C 90.000,E1 230.070} C_DIS
LIN {X 0.079,Y -152.112,Z 717.253,A 0.000,B 0.000,C 90.000,E1 225.567} C_DIS
LIN {X -0.014,Y -150.362,Z 717.238,A 0.000,B 0.000,C 90.000,E1 222.894} C_DIS
LIN {X 0.025,Y -147.097,Z 717.213,A 0.000,B 0.000,C 90.000,E1 218.338} C_DIS
LIN {X 0.020,Y -145.667,Z 717.198,A 0.000,B 0.000,C 90.000,E1 215.598} C_DIS
LIN {X 0.023,Y -143.049,Z 717.172,A 0.000,B 0.000,C 90.000,E1 211.003} C_DIS
LIN {X -0.042,Y -141.672,Z 717.152,A 0.000,B 0.000,C 90.000,E1 207.334} C_DIS
LIN {X 0.067,Y -139.452,Z 717.116,A 0.000,B 0.000,C 90.000,E1 200.791} C_DIS
LIN {X -0.012,Y -139.187,Z 717.105,A 0.000,B 0.000,C 90.000,E1 198.960} C_DIS
LIN {X 0.011,Y -138.322,Z 717.053,A 0.000,B 0.000,C 90.000,E1 189.613} C_DIS
LIN {X 0.018,Y -139.459,Z 717.007,A 0.000,B 0.000,C 90.000,E1 181.203} C_DIS
LIN {X -0.042,Y -141.014,Z 716.976,A 0.000,B 0.000,C 90.000,E1 175.641} C_DIS
LIN {X 0.049,Y -142.767,Z 716.955,A 0.000,B 0.000,C 90.000,E1 171.894} C_DIS
LIN {X 0.004,Y -145.178,Z 716.929,A 0.000,B 0.000,C 90.000,E1 167.297} C_DIS
LIN {X 0.038,Y -147.800,Z 716.909,A 0.000,B 0.000,C 90.000,E1 163.614} C_DIS
LIN {X -0.068,Y -150.484,Z 716.889,A 0.000,B 0.000,C 90.000,E1 160.007} C_DIS
LIN {X 0.006,Y -153.940,Z 716.869,A 0.000,B 0.000,C 90.000,E1 156.357} C_DIS
LIN {X 0.069,Y -157.350,Z 716.849,A 0.000,B 0.000,C 90.000,E1 152.743} C_DIS
LIN {X 0.012,Y -161.546,Z 716.829,A 0.000,B 0.000,C 90.000,E1 149.203} C_DIS
LIN {X 0.025,Y -165.744,Z 716.809,A 0.000,B 0.000,C 90.000,E1 145.674} C_DIS
LIN {X 0.012,Y -170.697,Z 716.790,A 0.000,B 0.000,C 90.000,E1 142.190} C_DIS
LIN {X -0.076,Y -175.571,Z 716.771,A 0.000,B 0.000,C 90.000,E1 138.771} C_DIS
LIN {X 0.043,Y -181.189,Z 716.752,A 0.000,B 0.000,C 90.000,E1 135.324} C_DIS
LIN {X -0.089,Y -186.650,Z 716.733,A 0.000,B 0.000,C 90.000,E1 132.000} C_DIS
LIN {X -0.020,Y -191.517,Z 716.718,A 0.000,B 0.000,C 90.000,E1 129.322} C_DIS
LIN {X 0.160,Y -289.900,Z 716.718,A 0.000,B 0.000,C 90.000,E1 129.277} C_DIS
LIN {X -0.044,Y -292.157,Z 716.718,A 0.000,B 0.000,C 90.000,E1 129.277} C_DIS
LIN {X 0.025,Y -297.590,Z 716.716,A 0.000,B 0.000,C 90.000,E1 128.955} C_DIS
LIN {X -0.093,Y -300.485,Z 716.715,A 0.000,B 0.000,C 90.000,E1 128.669} C_DIS
LIN {X -0.156,Y -302.519,Z 716.713,A 0.000,B 0.000,C 90.000,E1 128.382} C_DIS
LIN {X 0.019,Y -304.113,Z 716.711,A 0.000,B 0.000,C 90.000,E1 128.051} C_DIS
LIN {X -0.022,Y -305.509,Z 716.710,A 0.000,B 0.000,C 90.000,E1 127.729} C_DIS
LIN {X -0.008,Y -306.607,Z 716.708,A 0.000,B 0.000,C 90.000,E1 127.397} C_DIS
LIN {X 0.104,Y -316.273,Z 716.690,A 0.000,B 0.000,C 90.000,E1 124.119} C_DIS
LIN {X 0.002,Y -326.250,Z 716.674,A 0.000,B 0.000,C 90.000,E1 121.258} C_DIS
LIN {X -0.038,Y -337.551,Z 716.658,A 0.000,B 0.000,C 90.000,E1 118.437} C_DIS
LIN {X -0.060,Y -350.271,Z 716.643,A 0.000,B 0.000,C 90.000,E1 115.668} C_DIS
LIN {X -0.096,Y -362.865,Z 716.629,A 0.000,B 0.000,C 90.000,E1 113.259} C_DIS
LIN {X 0.097,Y -376.762,Z 716.616,A 0.000,B 0.000,C 90.000,E1 110.865} C_DIS
LIN {X 0.169,Y -392.063,Z 716.603,A 0.000,B 0.000,C 90.000,E1 108.544} C_DIS
LIN {X -0.016,Y -408.879,Z 716.591,A 0.000,B 0.000,C 90.000,E1 106.315} C_DIS
LIN {X -0.030,Y -427.330,Z 716.578,A 0.000,B 0.000,C 90.000,E1 104.120} C_DIS
LIN {X 0.062,Y -447.195,Z 716.567,A 0.000,B 0.000,C 90.000,E1 102.007} C_DIS
LIN {X 0.086,Y -467.667,Z 716.556,A 0.000,B 0.000,C 90.000,E1 100.074} C_DIS
LIN {X 0.044,Y -469.895,Z 716.555,A 0.000,B 0.000,C 90.000,E1 99.849} C_DIS
LIN {X -0.099,Y -471.716,Z 716.553,A 0.000,B 0.000,C 90.000,E1 99.613} C_DIS
LIN {X 0.224,Y -473.084,Z 716.552,A 0.000,B 0.000,C 90.000,E1 99.321} C_DIS
LIN {X -0.136,Y -474.816,Z 716.549,A 0.000,B 0.000,C 90.000,E1 98.859} C_DIS
LIN {X -0.017,Y -475.470,Z 716.546,A 0.000,B 0.000,C 90.000,E1 98.341} C_DIS
LIN {X 0.180,Y -475.158,Z 716.544,A 0.000,B 0.000,C 90.000,E1 97.814} C_DIS
LIN {X -0.158,Y -473.835,Z 716.541,A 0.000,B 0.000,C 90.000,E1 97.352} C_DIS
LIN {X 0.114,Y -472.729,Z 716.539,A 0.000,B 0.000,C 90.000,E1 97.068} C_DIS
LIN {X -0.227,Y -469.565,Z 716.537,A 0.000,B 0.000,C 90.000,E1 96.606} C_DIS
LIN {X 0.120,Y -453.297,Z 716.522,A 0.000,B 0.000,C 90.000,E1 94.012} C_DIS
LIN {X -0.099,Y -438.490,Z 716.508,A 0.000,B 0.000,C 90.000,E1 91.432} C_DIS
LIN {X -0.005,Y -429.480,Z 716.499,A 0.000,B 0.000,C 90.000,E1 89.828} C_DIS
LIN {X 0.058,Y -418.638,Z 716.489,A 0.000,B 0.000,C 90.000,E1 87.936} C_DIS
LIN {X -0.109,Y -407.649,Z 716.478,A 0.000,B 0.000,C 90.000,E1 86.045} C_DIS
LIN {X -0.043,Y -396.654,Z 716.467,A 0.000,B 0.000,C 90.000,E1 84.090} C_DIS
LIN {X -0.086,Y -379.602,Z 716.450,A 0.000,B 0.000,C 90.000,E1 80.971} C_DIS
LIN {X -0.009,Y -367.692,Z 716.437,A 0.000,B 0.000,C 90.000,E1 78.634} C_DIS
LIN {X 0.172,Y -354.846,Z 716.422,A 0.000,B 0.000,C 90.000,E1 75.936} C_DIS
LIN {X -0.088,Y -343.731,Z 716.409,A 0.000,B 0.000,C 90.000,E1 73.559} C_DIS
LIN {X -0.102,Y -331.533,Z 716.393,A 0.000,B 0.000,C 90.000,E1 70.786} C_DIS
LIN {X 0.015,Y -318.803,Z 716.376,A 0.000,B 0.000,C 90.000,E1 67.614} C_DIS
LIN {X 0.030,Y -308.666,Z 716.360,A 0.000,B 0.000,C 90.000,E1 64.717} C_DIS
LIN {X 0.089,Y -298.645,Z 716.341,A 0.000,B 0.000,C 90.000,E1 61.435} C_DIS
LIN {X 0.010,Y -289.261,Z 716.323,A 0.000,B 0.000,C 90.000,E1 58.122} C_DIS
LIN {X -0.146,Y -280.414,Z 716.304,A 0.000,B 0.000,C 90.000,E1 54.769} C_DIS
LIN {X -0.011,Y -275.242,Z 716.293,A 0.000,B 0.000,C 90.000,E1 52.683} C_DIS
LIN {X 0.024,Y -269.977,Z 716.281,A 0.000,B 0.000,C 90.000,E1 50.598} C_DIS
LIN {X 0.085,Y -264.508,Z 716.269,A 0.000,B 0.000,C 90.000,E1 48.485} C_DIS
LIN {X 0.023,Y -258.857,Z 716.258,A 0.000,B 0.000,C 90.000,E1 46.377} C_DIS
LIN {X -0.143,Y -253.102,Z 716.246,A 0.000,B 0.000,C 90.000,E1 44.271} C_DIS
LIN {X -0.050,Y -247.196,Z 716.234,A 0.000,B 0.000,C 90.000,E1 42.081} C_DIS
LIN {X 0.090,Y -239.096,Z 716.217,A 0.000,B 0.000,C 90.000,E1 39.116} C_DIS
LIN {X 0.056,Y -229.492,Z 716.197,A 0.000,B 0.000,C 90.000,E1 35.391} C_DIS
LIN {X 0.028,Y -220.647,Z 716.176,A 0.000,B 0.000,C 90.000,E1 31.592} C_DIS
LIN {X 0.067,Y -214.322,Z 716.158,A 0.000,B 0.000,C 90.000,E1 28.487} C_DIS
LIN {X 0.123,Y -208.821,Z 716.141,A 0.000,B 0.000,C 90.000,E1 25.335} C_DIS
LIN {X -0.033,Y -204.110,Z 716.123,A 0.000,B 0.000,C 90.000,E1 22.206} C_DIS
LIN {X 0.017,Y -199.240,Z 716.101,A 0.000,B 0.000,C 90.000,E1 18.181} C_DIS
LIN {X 0.052,Y -195.455,Z 716.079,A 0.000,B 0.000,C 90.000,E1 14.120} C_DIS
LIN {X 0.079,Y -192.377,Z 716.051,A 0.000,B 0.000,C 90.000,E1 9.208} C_DIS
LIN {X 0.050,Y -193.089,Z 715.961,A 0.000,B 0.000,C 90.000,E1 352.932} C_DIS
LIN {X -0.049,Y -196.450,Z 715.934,A 0.000,B 0.000,C 90.000,E1 348.049} C_DIS
LIN {X -0.012,Y -200.326,Z 715.911,A 0.000,B 0.000,C 90.000,E1 343.976} C_DIS
LIN {X 0.044,Y -205.205,Z 715.889,A 0.000,B 0.000,C 90.000,E1 339.934} C_DIS
LIN {X -0.035,Y -210.908,Z 715.866,A 0.000,B 0.000,C 90.000,E1 335.973} C_DIS
LIN {X 0.025,Y -217.351,Z 715.845,A 0.000,B 0.000,C 90.000,E1 332.025} C_DIS
LIN {X 0.125,Y -224.434,Z 715.823,A 0.000,B 0.000,C 90.000,E1 328.122} C_DIS
LIN {X 0.051,Y -232.109,Z 715.802,A 0.000,B 0.000,C 90.000,E1 324.322} C_DIS
LIN {X 0.065,Y -240.461,Z 715.781,A 0.000,B 0.000,C 90.000,E1 320.561} C_DIS
LIN {X -0.096,Y -249.690,Z 715.760,A 0.000,B 0.000,C 90.000,E1 316.905} C_DIS
LIN {X -0.004,Y -258.946,Z 715.742,A 0.000,B 0.000,C 90.000,E1 313.623} C_DIS
LIN {X -0.097,Y -270.242,Z 715.723,A 0.000,B 0.000,C 90.000,E1 310.092} C_DIS
LIN {X 0.077,Y -282.856,Z 715.703,A 0.000,B 0.000,C 90.000,E1 306.583} C_DIS
LIN {X -0.016,Y -296.861,Z 715.685,A 0.000,B 0.000,C 90.000,E1 303.214} C_DIS
LIN {X -0.068,Y -312.422,Z 715.666,A 0.000,B 0.000,C 90.000,E1 299.922} C_DIS
LIN {X 0.054,Y -329.696,Z 715.648,A 0.000,B 0.000,C 90.000,E1 296.693} C_DIS
LIN {X 0.011,Y -348.560,Z 715.631,A 0.000,B 0.000,C 90.000,E1 293.590} C_DIS
LIN {X 0.004,Y -364.575,Z 715.618,A 0.000,B 0.000,C 90.000,E1 291.173} C_DIS
LIN {X 0.149,Y -379.528,Z 715.606,A 0.000,B 0.000,C 90.000,E1 289.087} C_DIS
LIN {X 0.056,Y -398.061,Z 715.593,A 0.000,B 0.000,C 90.000,E1 286.804} C_DIS
LIN {X -0.026,Y -412.103,Z 715.584,A 0.000,B 0.000,C 90.000,E1 285.134} C_DIS
LIN {X 0.039,Y -425.767,Z 715.575,A 0.000,B 0.000,C 90.000,E1 283.480} C_DIS
LIN {X 0.161,Y -437.004,Z 715.567,A 0.000,B 0.000,C 90.000,E1 282.119} C_DIS
LIN {X 0.038,Y -445.509,Z 715.562,A 0.000,B 0.000,C 90.000,E1 281.074} C_DIS
LIN {X 0.087,Y -457.704,Z 715.553,A 0.000,B 0.000,C 90.000,E1 279.500} C_DIS
LIN {X 0.045,Y -467.673,Z 715.546,A 0.000,B 0.000,C 90.000,E1 278.219} C_DIS
LIN {X -0.034,Y -473.338,Z 715.541,A 0.000,B 0.000,C 90.000,E1 277.466} C_DIS
LIN {X -0.127,Y -478.340,Z 715.537,A 0.000,B 0.000,C 90.000,E1 276.720} C_DIS
LIN {X 0.017,Y -481.244,Z 715.534,A 0.000,B 0.000,C 90.000,E1 276.201} C_DIS
LIN {X 0.180,Y -483.704,Z 715.532,A 0.000,B 0.000,C 90.000,E1 275.682} C_DIS
LIN {X -0.125,Y -485.688,Z 715.529,A 0.000,B 0.000,C 90.000,E1 275.220} C_DIS
LIN {X 0.059,Y -487.344,Z 715.526,A 0.000,B 0.000,C 90.000,E1 274.702} C_DIS
LIN {X 0.217,Y -488.531,Z 715.523,A 0.000,B 0.000,C 90.000,E1 274.188} C_DIS
LIN {X -0.067,Y -489.325,Z 715.521,A 0.000,B 0.000,C 90.000,E1 273.726} C_DIS
LIN {X 0.113,Y -489.681,Z 715.518,A 0.000,B 0.000,C 90.000,E1 273.212} C_DIS
LIN {X -0.164,Y -489.706,Z 715.515,A 0.000,B 0.000,C 90.000,E1 272.751} C_DIS
LIN {X 0.027,Y -489.419,Z 715.512,A 0.000,B 0.000,C 90.000,E1 272.236} C_DIS
LIN {X 0.234,Y -488.758,Z 715.510,A 0.000,B 0.000,C 90.000,E1 271.718} C_DIS
LIN {X -0.065,Y -487.789,Z 715.507,A 0.000,B 0.000,C 90.000,E1 271.260} C_DIS
LIN {X 0.122,Y -486.459,Z 715.504,A 0.000,B 0.000,C 90.000,E1 270.745} C_DIS
LIN {X -0.182,Y -484.577,Z 715.501,A 0.000,B 0.000,C 90.000,E1 270.286} C_DIS
LIN {X -0.008,Y -482.146,Z 715.499,A 0.000,B 0.000,C 90.000,E1 269.771} C_DIS
LIN {X 0.147,Y -479.004,Z 715.496,A 0.000,B 0.000,C 90.000,E1 269.255} C_DIS
LIN {X -0.192,Y -475.102,Z 715.493,A 0.000,B 0.000,C 90.000,E1 268.797} C_DIS
LIN {X 0.102,Y -472.817,Z 715.492,A 0.000,B 0.000,C 90.000,E1 268.511} C_DIS
LIN {X -0.175,Y -467.461,Z 715.489,A 0.000,B 0.000,C 90.000,E1 268.051} C_DIS
LIN {X 0.178,Y -464.301,Z 715.488,A 0.000,B 0.000,C 90.000,E1 267.764} C_DIS
LIN {X -0.120,Y -461.222,Z 715.487,A 0.000,B 0.000,C 90.000,E1 267.593} C_DIS
LIN {X 0.044,Y -457.731,Z 715.485,A 0.000,B 0.000,C 90.000,E1 267.364} C_DIS
LIN {X 0.033,Y -450.652,Z 715.483,A 0.000,B 0.000,C 90.000,E1 267.020} C_DIS
LIN {X 0.115,Y -443.047,Z 715.482,A 0.000,B 0.000,C 90.000,E1 266.731} C_DIS
LIN {X -0.187,Y -434.700,Z 715.481,A 0.000,B 0.000,C 90.000,E1 266.560} C_DIS
LIN {X 0.122,Y -430.884,Z 715.480,A 0.000,B 0.000,C 90.000,E1 266.445} C_DIS
LIN {X -0.169,Y -423.044,Z 715.480,A 0.000,B 0.000,C 90.000,E1 266.388} C_DIS
LIN {X 0.083,Y -417.864,Z 715.480,A 0.000,B 0.000,C 90.000,E1 266.331} C_DIS
LIN {X 0.000,Y -180.937,Z 715.480,A 0.000,B 0.000,C 90.000,E1 266.331} C_DIS
LIN {X 0.007,Y -180.729,Z 715.470,A 0.000,B 0.000,C 90.000,E1 264.609} C_DIS
LIN {X -0.071,Y -178.818,Z 715.442,A 0.000,B 0.000,C 90.000,E1 259.567} C_DIS
LIN {X 0.011,Y -175.864,Z 715.414,A 0.000,B 0.000,C 90.000,E1 254.448} C_DIS
LIN {X 0.060,Y -173.830,Z 715.399,A 0.000,B 0.000,C 90.000,E1 251.873} C_DIS
LIN {X -0.005,Y -171.498,Z 715.380,A 0.000,B 0.000,C 90.000,E1 248.465} C_DIS
LIN {X -0.018,Y -167.726,Z 715.356,A 0.000,B 0.000,C 90.000,E1 244.152} C_DIS
LIN {X -0.002,Y -166.421,Z 715.347,A 0.000,B 0.000,C 90.000,E1 242.410} C_DIS
LIN {X -0.004,Y -163.142,Z 715.327,A 0.000,B 0.000,C 90.000,E1 238.918} C_DIS
LIN {X -0.038,Y -161.096,Z 715.313,A 0.000,B 0.000,C 90.000,E1 236.294} C_DIS
LIN {X -0.054,Y -157.824,Z 715.293,A 0.000,B 0.000,C 90.000,E1 232.763} C_DIS
LIN {X 0.009,Y -155.858,Z 715.278,A 0.000,B 0.000,C 90.000,E1 230.070} C_DIS
LIN {X 0.065,Y -152.108,Z 715.253,A 0.000,B 0.000,C 90.000,E1 225.567} C_DIS
LIN {X -0.027,Y -150.359,Z 715.238,A 0.000,B 0.000,C 90.000,E1 222.894} C_DIS
LIN {X 0.012,Y -147.094,Z 715.213,A 0.000,B 0.000,C 90.000,E1 218.338} C_DIS
LIN {X 0.006,Y -145.665,Z 715.198,A 0.000,B 0.000,C 90.000,E1 215.598} C_DIS
LIN {X 0.009,Y -143.046,Z 715.172,A 0.000,B 0.000,C 90.000,E1 211.003} C_DIS
LIN {X 0.010,Y -141.670,Z 715.152,A 0.000,B 0.000,C 90.000,E1 207.308} C_DIS
LIN {X 0.054,Y -139.452,Z 715.116,A 0.000,B 0.000,C 90.000,E1 200.791} C_DIS
LIN {X -0.024,Y -139.186,Z 715.105,A 0.000,B 0.000,C 90.000,E1 198.960} C_DIS
LIN {X -0.002,Y -138.322,Z 715.053,A 0.000,B 0.000,C 90.000,E1 189.613} C_DIS
LIN {X 0.005,Y -139.460,Z 715.007,A 0.000,B 0.000,C 90.000,E1 181.203} C_DIS
LIN {X -0.055,Y -141.016,Z 714.976,A 0.000,B 0.000,C 90.000,E1 175.641} C_DIS
LIN {X 0.036,Y -142.770,Z 714.955,A 0.000,B 0.000,C 90.000,E1 171.894} C_DIS
LIN {X -0.009,Y -145.180,Z 714.929,A 0.000,B 0.000,C 90.000,E1 167.297} C_DIS
LIN {X 0.024,Y -147.803,Z 714.909,A 0.000,B 0.000,C 90.000,E1 163.614} C_DIS
LIN {X -0.081,Y -150.489,Z 714.889,A 0.000,B 0.000,C 90.000,E1 160.007} C_DIS
LIN {X -0.008,Y -153.945,Z 714.869,A 0.000,B 0.000,C 90.000,E1 156.357} C_DIS
LIN {X 0.055,Y -157.356,Z 714.849,A 0.000,B 0.000,C 90.000,E1 152.743} C_DIS
LIN {X -0.001,Y -161.552,Z 714.829,A 0.000,B 0.000,C 90.000,E1 149.203} C_DIS
LIN {X 0.010,Y -165.750,Z 714.809,A 0.000,B 0.000,C 90.000,E1 145.674} C_DIS
LIN {X -0.003,Y -170.705,Z 714.790,A 0.000,B 0.000,C 90.000,E1 142.190} C_DIS
LIN {X -0.092,Y -175.579,Z 714.771,A 0.000,B 0.000,C 90.000,E1 138.771} C_DIS
LIN {X 0.028,Y -181.196,Z 714.752,A 0.000,B 0.000,C 90.000,E1 135.324} C_DIS
LIN {X 0.021,Y -186.657,Z 714.733,A 0.000,B 0.000,C 90.000,E1 131.962} C_DIS
LIN {X 0.011,Y -191.502,Z 714.718,A 0.000,B 0.000,C 90.000,E1 129.322} C_DIS
LIN {X -0.018,Y -290.269,Z 714.718,A 0.000,B 0.000,C 90.000,E1 129.322} C_DIS
LIN {X -0.068,Y -292.663,Z 714.718,A 0.000,B 0.000,C 90.000,E1 129.277} C_DIS
LIN {X 0.001,Y -297.734,Z 714.716,A 0.000,B 0.000,C 90.000,E1 128.955} C_DIS
LIN {X -0.118,Y -300.566,Z 714.715,A 0.000,B 0.000,C 90.000,E1 128.669} C_DIS
LIN {X 0.029,Y -302.599,Z 714.713,A 0.000,B 0.000,C 90.000,E1 128.338} C_DIS
LIN {X 0.128,Y -304.188,Z 714.711,A 0.000,B 0.000,C 90.000,E1 128.016} C_DIS
LIN {X -0.100,Y -305.556,Z 714.709,A 0.000,B 0.000,C 90.000,E1 127.729} C_DIS
LIN {X 0.100,Y -306.632,Z 714.708,A 0.000,B 0.000,C 90.000,E1 127.363} C_DIS
LIN {X 0.023,Y -316.299,Z 714.690,A 0.000,B 0.000,C 90.000,E1 124.119} C_DIS
LIN {X -0.080,Y -326.283,Z 714.674,A 0.000,B 0.000,C 90.000,E1 121.258} C_DIS
LIN {X 0.040,Y -337.589,Z 714.658,A 0.000,B 0.000,C 90.000,E1 118.409} C_DIS
LIN {X 0.005,Y -350.317,Z 714.642,A 0.000,B 0.000,C 90.000,E1 115.643} C_DIS
LIN {X 0.150,Y -362.918,Z 714.629,A 0.000,B 0.000,C 90.000,E1 113.206} C_DIS
LIN {X 0.008,Y -376.823,Z 714.616,A 0.000,B 0.000,C 90.000,E1 110.865} C_DIS
LIN {X 0.077,Y -392.131,Z 714.603,A 0.000,B 0.000,C 90.000,E1 108.544} C_DIS
LIN {X -0.111,Y -408.955,Z 714.591,A 0.000,B 0.000,C 90.000,E1 106.315} C_DIS
LIN {X -0.126,Y -427.417,Z 714.578,A 0.000,B 0.000,C 90.000,E1 104.120} C_DIS
LIN {X -0.031,Y -447.287,Z 714.567,A 0.000,B 0.000,C 90.000,E1 102.007} C_DIS
LIN {X -0.005,Y -467.762,Z 714.556,A 0.000,B 0.000,C 90.000,E1 100.074} C_DIS
LIN {X -0.047,Y -469.975,Z 714.555,A 0.000,B 0.000,C 90.000,E1 99.849} C_DIS
LIN {X -0.197,Y -471.791,Z 714.553,A 0.000,B 0.000,C 90.000,E1 99.613} C_DIS
LIN {X 0.117,Y -473.154,Z 714.552,A 0.000,B 0.000,C 90.000,E1 99.321} C_DIS
LIN {X -0.242,Y -474.870,Z 714.549,A 0.000,B 0.000,C 90.000,E1 98.859} C_DIS
LIN {X -0.123,Y -475.511,Z 714.546,A 0.000,B 0.000,C 90.000,E1 98.341} C_DIS
LIN {X 0.074,Y -475.185,Z 714.543,A 0.000,B 0.000,C 90.000,E1 97.814} C_DIS
LIN {X 0.207,Y -473.846,Z 714.541,A 0.000,B 0.000,C 90.000,E1 97.296} C_DIS
LIN {X 0.008,Y -472.733,Z 714.539,A 0.000,B 0.000,C 90.000,E1 97.068} C_DIS
LIN {X 0.135,Y -469.553,Z 714.536,A 0.000,B 0.000,C 90.000,E1 96.549} C_DIS
LIN {X 0.019,Y -453.285,Z 714.522,A 0.000,B 0.000,C 90.000,E1 94.012} C_DIS
LIN {X -0.197,Y -438.492,Z 714.508,A 0.000,B 0.000,C 90.000,E1 91.432} C_DIS
LIN {X 0.045,Y -427.934,Z 714.497,A 0.000,B 0.000,C 90.000,E1 89.542} C_DIS
LIN {X 0.070,Y -417.054,Z 714.487,A 0.000,B 0.000,C 90.000,E1 87.650} C_DIS
LIN {X -0.100,Y -406.073,Z 714.476,A 0.000,B 0.000,C 90.000,E1 85.755} C_DIS
LIN {X -0.064,Y -395.056,Z 714.466,A 0.000,B 0.000,C 90.000,E1 83.799} C_DIS
LIN {X -0.171,Y -379.644,Z 714.450,A 0.000,B 0.000,C 90.000,E1 80.971} C_DIS
LIN {X -0.090,Y -367.750,Z 714.437,A 0.000,B 0.000,C 90.000,E1 78.634} C_DIS
LIN {X 0.096,Y -354.911,Z 714.422,A 0.000,B 0.000,C 90.000,E1 75.936} C_DIS
LIN {X -0.160,Y -343.814,Z 714.409,A 0.000,B 0.000,C 90.000,E1 73.559} C_DIS
LIN {X 0.143,Y -331.651,Z 714.393,A 0.000,B 0.000,C 90.000,E1 70.732} C_DIS
LIN {X 0.021,Y -317.777,Z 714.374,A 0.000,B 0.000,C 90.000,E1 67.283} C_DIS
LIN {X -0.025,Y -308.852,Z 714.359,A 0.000,B 0.000,C 90.000,E1 64.717} C_DIS
LIN {X 0.042,Y -298.866,Z 714.341,A 0.000,B 0.000,C 90.000,E1 61.435} C_DIS
LIN {X -0.028,Y -289.510,Z 714.323,A 0.000,B 0.000,C 90.000,E1 58.122} C_DIS
LIN {X -0.013,Y -280.693,Z 714.304,A 0.000,B 0.000,C 90.000,E1 54.736} C_DIS
LIN {X -0.034,Y -275.534,Z 714.293,A 0.000,B 0.000,C 90.000,E1 52.683} C_DIS
LIN {X 0.006,Y -270.287,Z 714.281,A 0.000,B 0.000,C 90.000,E1 50.598} C_DIS
LIN {X 0.074,Y -264.826,Z 714.269,A 0.000,B 0.000,C 90.000,E1 48.485} C_DIS
LIN {X 0.018,Y -259.180,Z 714.258,A 0.000,B 0.000,C 90.000,E1 46.377} C_DIS
LIN {X -0.143,Y -253.403,Z 714.246,A 0.000,B 0.000,C 90.000,E1 44.271} C_DIS
LIN {X -0.044,Y -247.480,Z 714.234,A 0.000,B 0.000,C 90.000,E1 42.081} C_DIS
LIN {X 0.101,Y -239.377,Z 714.217,A 0.000,B 0.000,C 90.000,E1 39.116} C_DIS
LIN {X -0.034,Y -231.579,Z 714.201,A 0.000,B 0.000,C 90.000,E1 36.171} C_DIS
LIN {X 0.130,Y -222.559,Z 714.180,A 0.000,B 0.000,C 90.000,E1 32.339} C_DIS
LIN {X 0.028,Y -216.008,Z 714.163,A 0.000,B 0.000,C 90.000,E1 29.283} C_DIS
LIN {X 0.038,Y -210.299,Z 714.145,A 0.000,B 0.000,C 90.000,E1 26.155} C_DIS
LIN {X -0.081,Y -205.372,Z 714.128,A 0.000,B 0.000,C 90.000,E1 23.025} C_DIS
LIN {X -0.104,Y -200.255,Z 714.106,A 0.000,B 0.000,C 90.000,E1 19.033} C_DIS
LIN {X 0.024,Y -196.250,Z 714.083,A 0.000,B 0.000,C 90.000,E1 14.954} C_DIS
LIN {X -0.030,Y -192.913,Z 714.056,A 0.000,B 0.000,C 90.000,E1 10.074} C_DIS
LIN {X 0.029,Y -190.842,Z 714.010,A 0.000,B 0.000,C 90.000,E1 1.835} C_DIS
LIN {X 0.094,Y -192.812,Z 713.965,A 0.000,B 0.000,C 90.000,E1 353.742} C_DIS
LIN {X -0.053,Y -195.903,Z 713.938,A 0.000,B 0.000,C 90.000,E1 348.870} C_DIS
LIN {X -0.083,Y -199.588,Z 713.915,A 0.000,B 0.000,C 90.000,E1 344.810} C_DIS
LIN {X 0.077,Y -204.257,Z 713.893,A 0.000,B 0.000,C 90.000,E1 340.732} C_DIS
LIN {X 0.078,Y -209.798,Z 713.871,A 0.000,B 0.000,C 90.000,E1 336.741} C_DIS
LIN {X 0.002,Y -216.071,Z 713.849,A 0.000,B 0.000,C 90.000,E1 332.820} C_DIS
LIN {X -0.060,Y -223.003,Z 713.827,A 0.000,B 0.000,C 90.000,E1 328.948} C_DIS
LIN {X -0.001,Y -230.570,Z 713.806,A 0.000,B 0.000,C 90.000,E1 325.102} C_DIS
LIN {X 0.000,Y -238.764,Z 713.785,A 0.000,B 0.000,C 90.000,E1 321.331} C_DIS
LIN {X -0.025,Y -245.888,Z 713.769,A 0.000,B 0.000,C 90.000,E1 318.366} C_DIS
LIN {X -0.034,Y -255.779,Z 713.748,A 0.000,B 0.000,C 90.000,E1 314.717} C_DIS
LIN {X 0.086,Y -265.603,Z 713.731,A 0.000,B 0.000,C 90.000,E1 311.472} C_DIS
LIN {X -0.024,Y -276.417,Z 713.713,A 0.000,B 0.000,C 90.000,E1 308.338} C_DIS
LIN {X 0.019,Y -289.714,Z 713.694,A 0.000,B 0.000,C 90.000,E1 304.898} C_DIS
LIN {X 0.071,Y -304.454,Z 713.675,A 0.000,B 0.000,C 90.000,E1 301.544} C_DIS
LIN {X -0.033,Y -320.862,Z 713.657,A 0.000,B 0.000,C 90.000,E1 298.309} C_DIS
LIN {X -0.073,Y -338.893,Z 713.640,A 0.000,B 0.000,C 90.000,E1 295.155} C_DIS
LIN {X -0.019,Y -356.425,Z 713.624,A 0.000,B 0.000,C 90.000,E1 292.386} C_DIS
LIN {X 0.096,Y -377.144,Z 713.608,A 0.000,B 0.000,C 90.000,E1 289.396} C_DIS
LIN {X 0.106,Y -397.913,Z 713.593,A 0.000,B 0.000,C 90.000,E1 286.804} C_DIS
LIN {X 0.024,Y -411.922,Z 713.584,A 0.000,B 0.000,C 90.000,E1 285.134} C_DIS
LIN {X 0.088,Y -425.573,Z 713.575,A 0.000,B 0.000,C 90.000,E1 283.480} C_DIS
LIN {X 0.208,Y -436.813,Z 713.568,A 0.000,B 0.000,C 90.000,E1 282.119} C_DIS
LIN {X 0.083,Y -445.294,Z 713.562,A 0.000,B 0.000,C 90.000,E1 281.074} C_DIS
LIN {X 0.130,Y -457.473,Z 713.553,A 0.000,B 0.000,C 90.000,E1 279.500} C_DIS
LIN {X 0.084,Y -467.453,Z 713.546,A 0.000,B 0.000,C 90.000,E1 278.219} C_DIS
LIN {X 0.006,Y -473.132,Z 713.542,A 0.000,B 0.000,C 90.000,E1 277.466} C_DIS
LIN {X -0.089,Y -478.156,Z 713.537,A 0.000,B 0.000,C 90.000,E1 276.720} C_DIS
LIN {X -0.080,Y -482.363,Z 713.533,A 0.000,B 0.000,C 90.000,E1 275.967} C_DIS
LIN {X -0.089,Y -485.576,Z 713.529,A 0.000,B 0.000,C 90.000,E1 275.220} C_DIS
LIN {X 0.100,Y -487.213,Z 713.526,A 0.000,B 0.000,C 90.000,E1 274.702} C_DIS
LIN {X -0.230,Y -488.370,Z 713.523,A 0.000,B 0.000,C 90.000,E1 274.245} C_DIS
LIN {X -0.027,Y -489.184,Z 713.521,A 0.000,B 0.000,C 90.000,E1 273.726} C_DIS
LIN {X 0.152,Y -489.567,Z 713.518,A 0.000,B 0.000,C 90.000,E1 273.212} C_DIS
LIN {X -0.126,Y -489.591,Z 713.515,A 0.000,B 0.000,C 90.000,E1 272.751} C_DIS
LIN {X 0.063,Y -489.309,Z 713.512,A 0.000,B 0.000,C 90.000,E1 272.236} C_DIS
LIN {X -0.218,Y -488.617,Z 713.510,A 0.000,B 0.000,C 90.000,E1 271.776} C_DIS
LIN {X -0.029,Y -487.671,Z 713.507,A 0.000,B 0.000,C 90.000,E1 271.260} C_DIS
LIN {X 0.156,Y -486.348,Z 713.504,A 0.000,B 0.000,C 90.000,E1 270.745} C_DIS
LIN {X -0.148,Y -484.497,Z 713.501,A 0.000,B 0.000,C 90.000,E1 270.286} C_DIS
LIN {X 0.025,Y -482.064,Z 713.499,A 0.000,B 0.000,C 90.000,E1 269.771} C_DIS
LIN {X 0.179,Y -478.949,Z 713.496,A 0.000,B 0.000,C 90.000,E1 269.255} C_DIS
LIN {X -0.161,Y -475.065,Z 713.493,A 0.000,B 0.000,C 90.000,E1 268.797} C_DIS
LIN {X 0.134,Y -472.775,Z 713.492,A 0.000,B 0.000,C 90.000,E1 268.511} C_DIS
LIN {X -0.139,Y -467.441,Z 713.489,A 0.000,B 0.000,C 90.000,E1 268.051} C_DIS
LIN {X 0.218,Y -464.324,Z 713.488,A 0.000,B 0.000,C 90.000,E1 267.764} C_DIS
LIN {X -0.094,Y -461.244,Z 713.487,A 0.000,B 0.000,C 90.000,E1 267.593} C_DIS
LIN {X 0.058,Y -454.409,Z 713.484,A 0.000,B 0.000,C 90.000,E1 267.192} C_DIS
LIN {X -0.150,Y -447.256,Z 713.483,A 0.000,B 0.000,C 90.000,E1 266.906} C_DIS
LIN {X 0.184,Y -439.419,Z 713.481,A 0.000,B 0.000,C 90.000,E1 266.617} C_DIS
LIN {X 0.121,Y -431.139,Z 713.480,A 0.000,B 0.000,C 90.000,E1 266.445} C_DIS
LIN {X -0.008,Y -425.908,Z 713.480,A 0.000,B 0.000,C 90.000,E1 266.388} C_DIS
LIN {X -0.014,Y -416.562,Z 713.480,A 0.000,B 0.000,C 90.000,E1 266.331} C_DIS
LIN {X -0.027,Y -180.937,Z 713.480,A 0.000,B 0.000,C 90.000,E1 266.331} C_DIS
LIN {X -0.013,Y -180.727,Z 713.470,A 0.000,B 0.000,C 90.000,E1 264.609} C_DIS
LIN {X 0.084,Y -178.815,Z 713.442,A 0.000,B 0.000,C 90.000,E1 259.511} C_DIS
LIN {X -0.009,Y -175.860,Z 713.414,A 0.000,B 0.000,C 90.000,E1 254.448} C_DIS
LIN {X 0.040,Y -173.826,Z 713.399,A 0.000,B 0.000,C 90.000,E1 251.873} C_DIS
LIN {X -0.025,Y -171.492,Z 713.380,A 0.000,B 0.000,C 90.000,E1 248.465} C_DIS
LIN {X -0.038,Y -167.721,Z 713.356,A 0.000,B 0.000,C 90.000,E1 244.152} C_DIS
LIN {X -0.022,Y -166.413,Z 713.347,A 0.000,B 0.000,C 90.000,E1 242.410} C_DIS
LIN {X -0.024,Y -163.136,Z 713.327,A 0.000,B 0.000,C 90.000,E1 238.918} C_DIS
LIN {X -0.057,Y -161.089,Z 713.313,A 0.000,B 0.000,C 90.000,E1 236.294} C_DIS
LIN {X -0.073,Y -157.819,Z 713.293,A 0.000,B 0.000,C 90.000,E1 232.763} C_DIS
LIN {X -0.009,Y -155.853,Z 713.278,A 0.000,B 0.000,C 90.000,E1 230.070} C_DIS
LIN {X 0.046,Y -152.103,Z 713.253,A 0.000,B 0.000,C 90.000,E1 225.567} C_DIS
LIN {X 0.065,Y -150.354,Z 713.238,A 0.000,B 0.000,C 90.000,E1 222.852} C_DIS
LIN {X -0.006,Y -147.090,Z 713.213,A 0.000,B 0.000,C 90.000,E1 218.338} C_DIS
LIN {X -0.012,Y -145.661,Z 713.198,A 0.000,B 0.000,C 90.000,E1 215.598} C_DIS
LIN {X -0.008,Y -143.043,Z 713.172,A 0.000,B 0.000,C 90.000,E1 211.003} C_DIS
LIN {X -0.008,Y -141.668,Z 713.152,A 0.000,B 0.000,C 90.000,E1 207.308} C_DIS
LIN {X 0.037,Y -139.451,Z 713.116,A 0.000,B 0.000,C 90.000,E1 200.791} C_DIS
LIN {X -0.043,Y -139.185,Z 713.105,A 0.000,B 0.000,C 90.000,E1 198.960} C_DIS
LIN {X -0.019,Y -138.322,Z 713.053,A 0.000,B 0.000,C 90.000,E1 189.613} C_DIS
LIN {X -0.012,Y -139.461,Z 713.007,A 0.000,B 0.000,C 90.000,E1 181.203} C_DIS
LIN {X 0.068,Y -141.019,Z 712.976,A 0.000,B 0.000,C 90.000,E1 175.584} C_DIS
LIN {X 0.023,Y -142.382,Z 712.960,A 0.000,B 0.000,C 90.000,E1 172.818} C_DIS
LIN {X -0.056,Y -144.613,Z 712.935,A 0.000,B 0.000,C 90.000,E1 168.229} C_DIS
LIN {X 0.005,Y -147.807,Z 712.909,A 0.000,B 0.000,C 90.000,E1 163.614} C_DIS
LIN {X 0.041,Y -150.495,Z 712.889,A 0.000,B 0.000,C 90.000,E1 159.953} C_DIS
LIN {X -0.027,Y -153.952,Z 712.869,A 0.000,B 0.000,C 90.000,E1 156.357} C_DIS
LIN {X 0.035,Y -157.363,Z 712.849,A 0.000,B 0.000,C 90.000,E1 152.743} C_DIS
LIN {X -0.021,Y -161.562,Z 712.829,A 0.000,B 0.000,C 90.000,E1 149.203} C_DIS
LIN {X -0.010,Y -165.759,Z 712.809,A 0.000,B 0.000,C 90.000,E1 145.674} C_DIS
LIN {X -0.023,Y -170.716,Z 712.790,A 0.000,B 0.000,C 90.000,E1 142.190} C_DIS
LIN {X 0.020,Y -175.589,Z 712.771,A 0.000,B 0.000,C 90.000,E1 138.728} C_DIS
LIN {X 0.007,Y -181.206,Z 712.752,A 0.000,B 0.000,C 90.000,E1 135.324} C_DIS
LIN {X 0.000,Y -186.669,Z 712.733,A 0.000,B 0.000,C 90.000,E1 131.962} C_DIS
LIN {X -0.039,Y -191.467,Z 712.719,A 0.000,B 0.000,C 90.000,E1 129.358} C_DIS
LIN {X -0.111,Y -289.944,Z 712.719,A 0.000,B 0.000,C 90.000,E1 129.358} C_DIS
LIN {X 0.010,Y -295.227,Z 712.718,A 0.000,B 0.000,C 90.000,E1 129.152} C_DIS
LIN {X -0.043,Y -297.532,Z 712.717,A 0.000,B 0.000,C 90.000,E1 128.991} C_DIS
LIN {X 0.083,Y -300.667,Z 712.715,A 0.000,B 0.000,C 90.000,E1 128.624} C_DIS
LIN {X -0.008,Y -302.666,Z 712.713,A 0.000,B 0.000,C 90.000,E1 128.338} C_DIS
LIN {X 0.087,Y -304.232,Z 712.711,A 0.000,B 0.000,C 90.000,E1 128.016} C_DIS
LIN {X -0.141,Y -305.578,Z 712.709,A 0.000,B 0.000,C 90.000,E1 127.729} C_DIS
LIN {X 0.048,Y -308.452,Z 712.704,A 0.000,B 0.000,C 90.000,E1 126.710} C_DIS
LIN {X -0.154,Y -318.413,Z 712.686,A 0.000,B 0.000,C 90.000,E1 123.499} C_DIS
LIN {X 0.077,Y -328.684,Z 712.670,A 0.000,B 0.000,C 90.000,E1 120.590} C_DIS
LIN {X 0.109,Y -340.303,Z 712.654,A 0.000,B 0.000,C 90.000,E1 117.769} C_DIS
LIN {X 0.007,Y -353.365,Z 712.639,A 0.000,B 0.000,C 90.000,E1 115.027} C_DIS
LIN {X -0.098,Y -366.286,Z 712.626,A 0.000,B 0.000,C 90.000,E1 112.642} C_DIS
LIN {X -0.170,Y -380.536,Z 712.613,A 0.000,B 0.000,C 90.000,E1 110.301} C_DIS
LIN {X -0.149,Y -396.218,Z 712.600,A 0.000,B 0.000,C 90.000,E1 108.000} C_DIS
LIN {X 0.147,Y -413.445,Z 712.587,A 0.000,B 0.000,C 90.000,E1 105.717} C_DIS
LIN {X 0.153,Y -432.339,Z 712.575,A 0.000,B 0.000,C 90.000,E1 103.536} C_DIS
LIN {X 0.155,Y -452.394,Z 712.564,A 0.000,B 0.000,C 90.000,E1 101.478} C_DIS
LIN {X -0.055,Y -467.802,Z 712.556,A 0.000,B 0.000,C 90.000,E1 100.074} C_DIS
LIN {X -0.097,Y -470.015,Z 712.555,A 0.000,B 0.000,C 90.000,E1 99.849} C_DIS
LIN {X 0.218,Y -471.830,Z 712.553,A 0.000,B 0.000,C 90.000,E1 99.557} C_DIS
LIN {X 0.066,Y -473.194,Z 712.552,A 0.000,B 0.000,C 90.000,E1 99.321} C_DIS
LIN {X 0.176,Y -474.909,Z 712.549,A 0.000,B 0.000,C 90.000,E1 98.803} C_DIS
LIN {X -0.174,Y -475.550,Z 712.546,A 0.000,B 0.000,C 90.000,E1 98.341} C_DIS
LIN {X 0.023,Y -475.224,Z 712.543,A 0.000,B 0.000,C 90.000,E1 97.814} C_DIS
LIN {X 0.157,Y -473.885,Z 712.541,A 0.000,B 0.000,C 90.000,E1 97.296} C_DIS
LIN {X -0.042,Y -472.771,Z 712.539,A 0.000,B 0.000,C 90.000,E1 97.068} C_DIS
LIN {X 0.086,Y -469.586,Z 712.536,A 0.000,B 0.000,C 90.000,E1 96.549} C_DIS
LIN {X 0.191,Y -451.776,Z 712.521,A 0.000,B 0.000,C 90.000,E1 93.726} C_DIS
LIN {X 0.197,Y -438.520,Z 712.508,A 0.000,B 0.000,C 90.000,E1 91.375} C_DIS
LIN {X -0.143,Y -429.509,Z 712.499,A 0.000,B 0.000,C 90.000,E1 89.828} C_DIS
LIN {X -0.206,Y -420.214,Z 712.490,A 0.000,B 0.000,C 90.000,E1 88.224} C_DIS
LIN {X 0.094,Y -409.251,Z 712.479,A 0.000,B 0.000,C 90.000,E1 86.274} C_DIS
LIN {X 0.189,Y -398.263,Z 712.469,A 0.000,B 0.000,C 90.000,E1 84.318} C_DIS
LIN {X 0.168,Y -382.738,Z 712.453,A 0.000,B 0.000,C 90.000,E1 81.489} C_DIS
LIN {X -0.114,Y -369.313,Z 712.438,A 0.000,B 0.000,C 90.000,E1 78.926} C_DIS
LIN {X 0.112,Y -356.416,Z 712.424,A 0.000,B 0.000,C 90.000,E1 76.228} C_DIS
LIN {X 0.145,Y -343.942,Z 712.409,A 0.000,B 0.000,C 90.000,E1 73.504} C_DIS
LIN {X 0.105,Y -330.513,Z 712.391,A 0.000,B 0.000,C 90.000,E1 70.423} C_DIS
LIN {X 0.007,Y -317.972,Z 712.374,A 0.000,B 0.000,C 90.000,E1 67.283} C_DIS
LIN {X -0.033,Y -309.068,Z 712.359,A 0.000,B 0.000,C 90.000,E1 64.717} C_DIS
LIN {X 0.042,Y -299.107,Z 712.341,A 0.000,B 0.000,C 90.000,E1 61.435} C_DIS
LIN {X -0.021,Y -289.785,Z 712.323,A 0.000,B 0.000,C 90.000,E1 58.122} C_DIS
LIN {X -0.160,Y -280.995,Z 712.304,A 0.000,B 0.000,C 90.000,E1 54.769} C_DIS
LIN {X -0.014,Y -275.848,Z 712.293,A 0.000,B 0.000,C 90.000,E1 52.683} C_DIS
LIN {X 0.031,Y -270.608,Z 712.281,A 0.000,B 0.000,C 90.000,E1 50.598} C_DIS
LIN {X 0.105,Y -265.164,Z 712.269,A 0.000,B 0.000,C 90.000,E1 48.485} C_DIS
LIN {X 0.055,Y -259.531,Z 712.258,A 0.000,B 0.000,C 90.000,E1 46.377} C_DIS
LIN {X -0.101,Y -253.719,Z 712.246,A 0.000,B 0.000,C 90.000,E1 44.271} C_DIS
LIN {X 0.003,Y -247.776,Z 712.234,A 0.000,B 0.000,C 90.000,E1 42.081} C_DIS
LIN {X 0.004,Y -239.654,Z 712.218,A 0.000,B 0.000,C 90.000,E1 39.152} C_DIS
LIN {X 0.024,Y -231.821,Z 712.201,A 0.000,B 0.000,C 90.000,E1 36.171} C_DIS
LIN {X -0.114,Y -222.787,Z 712.180,A 0.000,B 0.000,C 90.000,E1 32.418} C_DIS
LIN {X -0.092,Y -216.215,Z 712.163,A 0.000,B 0.000,C 90.000,E1 29.333} C_DIS
LIN {X 0.015,Y -210.478,Z 712.145,A 0.000,B 0.000,C 90.000,E1 26.181} C_DIS
LIN {X -0.008,Y -205.535,Z 712.128,A 0.000,B 0.000,C 90.000,E1 23.025} C_DIS
LIN {X -0.028,Y -200.393,Z 712.106,A 0.000,B 0.000,C 90.000,E1 19.033} C_DIS
LIN {X -0.087,Y -196.392,Z 712.083,A 0.000,B 0.000,C 90.000,E1 15.009} C_DIS
LIN {X 0.052,Y -193.050,Z 712.056,A 0.000,B 0.000,C 90.000,E1 10.074} C_DIS
LIN {X -0.072,Y -190.968,Z 712.010,A 0.000,B 0.000,C 90.000,E1 1.892} C_DIS
LIN {X -0.092,Y -192.945,Z 711.965,A 0.000,B 0.000,C 90.000,E1 353.799} C_DIS
LIN {X -0.042,Y -196.011,Z 711.938,A 0.000,B 0.000,C 90.000,E1 348.870} C_DIS
LIN {X -0.068,Y -199.698,Z 711.916,A 0.000,B 0.000,C 90.000,E1 344.810} C_DIS
LIN {X 0.095,Y -204.358,Z 711.893,A 0.000,B 0.000,C 90.000,E1 340.732} C_DIS
LIN {X -0.093,Y -209.885,Z 711.871,A 0.000,B 0.000,C 90.000,E1 336.794} C_DIS
LIN {X 0.027,Y -216.127,Z 711.849,A 0.000,B 0.000,C 90.000,E1 332.820} C_DIS
LIN {X -0.032,Y -223.048,Z 711.827,A 0.000,B 0.000,C 90.000,E1 328.948} C_DIS
LIN {X 0.029,Y -230.609,Z 711.806,A 0.000,B 0.000,C 90.000,E1 325.102} C_DIS
LIN {X 0.032,Y -238.775,Z 711.785,A 0.000,B 0.000,C 90.000,E1 321.331} C_DIS
LIN {X 0.008,Y -245.905,Z 711.769,A 0.000,B 0.000,C 90.000,E1 318.366} C_DIS
LIN {X -0.007,Y -254.755,Z 711.750,A 0.000,B 0.000,C 90.000,E1 315.081} C_DIS
LIN {X -0.077,Y -265.610,Z 711.731,A 0.000,B 0.000,C 90.000,E1 311.515} C_DIS
LIN {X 0.015,Y -276.435,Z 711.713,A 0.000,B 0.000,C 90.000,E1 308.338} C_DIS
LIN {X 0.060,Y -289.752,Z 711.694,A 0.000,B 0.000,C 90.000,E1 304.898} C_DIS
LIN {X 0.116,Y -304.476,Z 711.675,A 0.000,B 0.000,C 90.000,E1 301.544} C_DIS
LIN {X 0.015,Y -320.866,Z 711.657,A 0.000,B 0.000,C 90.000,E1 298.309} C_DIS
LIN {X -0.023,Y -338.872,Z 711.640,A 0.000,B 0.000,C 90.000,E1 295.155} C_DIS
LIN {X 0.033,Y -356.355,Z 711.624,A 0.000,B 0.000,C 90.000,E1 292.386} C_DIS
LIN {X 0.041,Y -374.857,Z 711.609,A 0.000,B 0.000,C 90.000,E1 289.704} C_DIS
LIN {X 0.156,Y -397.765,Z 711.594,A 0.000,B 0.000,C 90.000,E1 286.804} C_DIS
LIN {X 0.074,Y -411.735,Z 711.584,A 0.000,B 0.000,C 90.000,E1 285.134} C_DIS
LIN {X 0.135,Y -425.392,Z 711.575,A 0.000,B 0.000,C 90.000,E1 283.480} C_DIS
LIN {X -0.174,Y -436.620,Z 711.568,A 0.000,B 0.000,C 90.000,E1 282.175} C_DIS
LIN {X -0.089,Y -447.152,Z 711.560,A 0.000,B 0.000,C 90.000,E1 280.838} C_DIS
LIN {X -0.197,Y -461.272,Z 711.550,A 0.000,B 0.000,C 90.000,E1 279.029} C_DIS
LIN {X 0.198,Y -471.081,Z 711.543,A 0.000,B 0.000,C 90.000,E1 277.701} C_DIS
LIN {X 0.152,Y -476.363,Z 711.539,A 0.000,B 0.000,C 90.000,E1 276.947} C_DIS
LIN {X 0.089,Y -480.874,Z 711.534,A 0.000,B 0.000,C 90.000,E1 276.201} C_DIS
LIN {X -0.230,Y -483.365,Z 711.532,A 0.000,B 0.000,C 90.000,E1 275.739} C_DIS
LIN {X -0.056,Y -485.420,Z 711.529,A 0.000,B 0.000,C 90.000,E1 275.220} C_DIS
LIN {X 0.133,Y -487.077,Z 711.526,A 0.000,B 0.000,C 90.000,E1 274.702} C_DIS
LIN {X -0.198,Y -488.278,Z 711.523,A 0.000,B 0.000,C 90.000,E1 274.245} C_DIS
LIN {X 0.004,Y -489.041,Z 711.521,A 0.000,B 0.000,C 90.000,E1 273.726} C_DIS
LIN {X 0.183,Y -489.461,Z 711.518,A 0.000,B 0.000,C 90.000,E1 273.212} C_DIS
LIN {X -0.095,Y -489.498,Z 711.515,A 0.000,B 0.000,C 90.000,E1 272.751} C_DIS
LIN {X 0.094,Y -489.178,Z 711.512,A 0.000,B 0.000,C 90.000,E1 272.236} C_DIS
LIN {X -0.188,Y -488.569,Z 711.510,A 0.000,B 0.000,C 90.000,E1 271.776} C_DIS
LIN {X 0.000,Y -487.588,Z 711.507,A 0.000,B 0.000,C 90.000,E1 271.260} C_DIS
LIN {X 0.184,Y -486.244,Z 711.504,A 0.000,B 0.000,C 90.000,E1 270.745} C_DIS
LIN {X -0.121,Y -484.422,Z 711.502,A 0.000,B 0.000,C 90.000,E1 270.286} C_DIS
LIN {X 0.052,Y -482.009,Z 711.499,A 0.000,B 0.000,C 90.000,E1 269.771} C_DIS
LIN {X 0.205,Y -478.945,Z 711.496,A 0.000,B 0.000,C 90.000,E1 269.255} C_DIS
LIN {X -0.135,Y -475.055,Z 711.493,A 0.000,B 0.000,C 90.000,E1 268.797} C_DIS
LIN {X -0.019,Y -470.198,Z 711.490,A 0.000,B 0.000,C 90.000,E1 268.282} C_DIS
LIN {X 0.186,Y -464.226,Z 711.488,A 0.000,B 0.000,C 90.000,E1 267.764} C_DIS
LIN {X -0.134,Y -461.092,Z 711.487,A 0.000,B 0.000,C 90.000,E1 267.593} C_DIS
LIN {X 0.005,Y -454.277,Z 711.484,A 0.000,B 0.000,C 90.000,E1 267.192} C_DIS
LIN {X -0.204,Y -447.125,Z 711.483,A 0.000,B 0.000,C 90.000,E1 266.906} C_DIS
LIN {X 0.133,Y -439.328,Z 711.481,A 0.000,B 0.000,C 90.000,E1 266.617} C_DIS
LIN {X 0.065,Y -431.047,Z 711.480,A 0.000,B 0.000,C 90.000,E1 266.445} C_DIS
LIN {X -0.072,Y -425.820,Z 711.480,A 0.000,B 0.000,C 90.000,E1 266.388} C_DIS
LIN {X -0.031,Y -419.371,Z 711.480,A 0.000,B 0.000,C 90.000,E1 266.331} C_DIS
LIN {X -0.034,Y -180.936,Z 711.480,A 0.000,B 0.000,C 90.000,E1 266.331} C_DIS
LIN {X -0.044,Y -180.722,Z 711.470,A 0.000,B 0.000,C 90.000,E1 264.609} C_DIS
LIN {X 0.054,Y -178.810,Z 711.442,A 0.000,B 0.000,C 90.000,E1 259.511} C_DIS
LIN {X -0.039,Y -175.855,Z 711.414,A 0.000,B 0.000,C 90.000,E1 254.448} C_DIS
LIN {X -0.057,Y -173.183,Z 711.395,A 0.000,B 0.000,C 90.000,E1 251.040} C_DIS
LIN {X -0.054,Y -171.484,Z 711.380,A 0.000,B 0.000,C 90.000,E1 248.465} C_DIS
LIN {X -0.067,Y -167.714,Z 711.356,A 0.000,B 0.000,C 90.000,E1 244.152} C_DIS
LIN {X -0.050,Y -166.404,Z 711.347,A 0.000,B 0.000,C 90.000,E1 242.410} C_DIS
LIN {X 0.088,Y -163.128,Z 711.327,A 0.000,B 0.000,C 90.000,E1 238.869} C_DIS
LIN {X -0.085,Y -161.079,Z 711.313,A 0.000,B 0.000,C 90.000,E1 236.294} C_DIS
LIN {X 0.024,Y -157.810,Z 711.293,A 0.000,B 0.000,C 90.000,E1 232.718} C_DIS
LIN {X -0.038,Y -155.845,Z 711.278,A 0.000,B 0.000,C 90.000,E1 230.070} C_DIS
LIN {X 0.018,Y -152.096,Z 711.253,A 0.000,B 0.000,C 90.000,E1 225.567} C_DIS
LIN {X 0.037,Y -150.347,Z 711.238,A 0.000,B 0.000,C 90.000,E1 222.852} C_DIS
LIN {X 0.058,Y -147.084,Z 711.213,A 0.000,B 0.000,C 90.000,E1 218.302} C_DIS
LIN {X -0.038,Y -145.656,Z 711.198,A 0.000,B 0.000,C 90.000,E1 215.598} C_DIS
LIN {X -0.035,Y -143.039,Z 711.172,A 0.000,B 0.000,C 90.000,E1 211.003} C_DIS
LIN {X -0.035,Y -141.663,Z 711.152,A 0.000,B 0.000,C 90.000,E1 207.308} C_DIS
LIN {X 0.011,Y -139.448,Z 711.116,A 0.000,B 0.000,C 90.000,E1 200.791} C_DIS
LIN {X 0.063,Y -139.182,Z 711.105,A 0.000,B 0.000,C 90.000,E1 198.906} C_DIS
LIN {X -0.045,Y -138.321,Z 711.053,A 0.000,B 0.000,C 90.000,E1 189.613} C_DIS
LIN {X -0.038,Y -139.463,Z 711.007,A 0.000,B 0.000,C 90.000,E1 181.203} C_DIS
LIN {X 0.042,Y -141.023,Z 710.976,A 0.000,B 0.000,C 90.000,E1 175.584} C_DIS
LIN {X -0.004,Y -142.389,Z 710.960,A 0.000,B 0.000,C 90.000,E1 172.818} C_DIS
LIN {X 0.059,Y -144.620,Z 710.934,A 0.000,B 0.000,C 90.000,E1 168.173} C_DIS
LIN {X -0.022,Y -147.814,Z 710.909,A 0.000,B 0.000,C 90.000,E1 163.614} C_DIS
LIN {X 0.066,Y -150.504,Z 710.889,A 0.000,B 0.000,C 90.000,E1 159.934} C_DIS
LIN {X -0.054,Y -153.962,Z 710.869,A 0.000,B 0.000,C 90.000,E1 156.357} C_DIS
LIN {X 0.007,Y -157.374,Z 710.849,A 0.000,B 0.000,C 90.000,E1 152.743} C_DIS
LIN {X -0.050,Y -161.575,Z 710.829,A 0.000,B 0.000,C 90.000,E1 149.203} C_DIS
LIN {X -0.038,Y -165.773,Z 710.809,A 0.000,B 0.000,C 90.000,E1 145.674} C_DIS
LIN {X -0.053,Y -170.731,Z 710.790,A 0.000,B 0.000,C 90.000,E1 142.190} C_DIS
LIN {X -0.010,Y -175.604,Z 710.771,A 0.000,B 0.000,C 90.000,E1 138.728} C_DIS
LIN {X -0.024,Y -181.220,Z 710.752,A 0.000,B 0.000,C 90.000,E1 135.324} C_DIS
LIN {X -0.032,Y -186.686,Z 710.733,A 0.000,B 0.000,C 90.000,E1 131.962} C_DIS
LIN {X -0.001,Y -191.449,Z 710.719,A 0.000,B 0.000,C 90.000,E1 129.358} C_DIS
LIN {X -0.054,Y -290.277,Z 710.719,A 0.000,B 0.000,C 90.000,E1 129.358} C_DIS
LIN {X -0.027,Y -291.843,Z 710.718,A 0.000,B 0.000,C 90.000,E1 129.322} C_DIS
LIN {X 0.148,Y -295.555,Z 710.717,A 0.000,B 0.000,C 90.000,E1 129.116} C_DIS
LIN {X -0.092,Y -297.747,Z 710.716,A 0.000,B 0.000,C 90.000,E1 128.991} C_DIS
LIN {X 0.033,Y -300.790,Z 710.715,A 0.000,B 0.000,C 90.000,E1 128.624} C_DIS
LIN {X 0.094,Y -302.784,Z 710.713,A 0.000,B 0.000,C 90.000,E1 128.302} C_DIS
LIN {X -0.036,Y -304.344,Z 710.711,A 0.000,B 0.000,C 90.000,E1 128.016} C_DIS
LIN {X -0.023,Y -305.653,Z 710.709,A 0.000,B 0.000,C 90.000,E1 127.684} C_DIS
LIN {X 0.169,Y -310.373,Z 710.700,A 0.000,B 0.000,C 90.000,E1 126.011} C_DIS
LIN {X -0.136,Y -320.641,Z 710.682,A 0.000,B 0.000,C 90.000,E1 122.832} C_DIS
LIN {X 0.000,Y -331.213,Z 710.666,A 0.000,B 0.000,C 90.000,E1 119.951} C_DIS
LIN {X 0.111,Y -343.154,Z 710.651,A 0.000,B 0.000,C 90.000,E1 117.129} C_DIS
LIN {X 0.091,Y -356.565,Z 710.636,A 0.000,B 0.000,C 90.000,E1 114.387} C_DIS
LIN {X -0.079,Y -369.821,Z 710.622,A 0.000,B 0.000,C 90.000,E1 112.025} C_DIS
LIN {X -0.063,Y -384.432,Z 710.609,A 0.000,B 0.000,C 90.000,E1 109.685} C_DIS
LIN {X -0.066,Y -400.502,Z 710.597,A 0.000,B 0.000,C 90.000,E1 107.402} C_DIS
LIN {X -0.169,Y -418.148,Z 710.584,A 0.000,B 0.000,C 90.000,E1 105.190} C_DIS
LIN {X -0.015,Y -437.448,Z 710.572,A 0.000,B 0.000,C 90.000,E1 103.008} C_DIS
LIN {X -0.106,Y -457.654,Z 710.561,A 0.000,B 0.000,C 90.000,E1 101.007} C_DIS
LIN {X -0.193,Y -467.960,Z 710.556,A 0.000,B 0.000,C 90.000,E1 100.074} C_DIS
LIN {X -0.235,Y -470.141,Z 710.555,A 0.000,B 0.000,C 90.000,E1 99.849} C_DIS
LIN {X 0.079,Y -471.936,Z 710.553,A 0.000,B 0.000,C 90.000,E1 99.557} C_DIS
LIN {X -0.073,Y -473.283,Z 710.552,A 0.000,B 0.000,C 90.000,E1 99.321} C_DIS
LIN {X 0.036,Y -474.972,Z 710.549,A 0.000,B 0.000,C 90.000,E1 98.803} C_DIS
LIN {X 0.226,Y -475.592,Z 710.546,A 0.000,B 0.000,C 90.000,E1 98.276} C_DIS
LIN {X -0.116,Y -475.245,Z 710.543,A 0.000,B 0.000,C 90.000,E1 97.814} C_DIS
LIN {X 0.018,Y -473.883,Z 710.541,A 0.000,B 0.000,C 90.000,E1 97.296} C_DIS
LIN {X -0.180,Y -472.754,Z 710.539,A 0.000,B 0.000,C 90.000,E1 97.068} C_DIS
LIN {X -0.051,Y -469.547,Z 710.536,A 0.000,B 0.000,C 90.000,E1 96.549} C_DIS
LIN {X 0.059,Y -451.736,Z 710.521,A 0.000,B 0.000,C 90.000,E1 93.726} C_DIS
LIN {X 0.067,Y -438.477,Z 710.508,A 0.000,B 0.000,C 90.000,E1 91.375} C_DIS
LIN {X 0.158,Y -429.479,Z 710.499,A 0.000,B 0.000,C 90.000,E1 89.771} C_DIS
LIN {X 0.102,Y -420.189,Z 710.490,A 0.000,B 0.000,C 90.000,E1 88.165} C_DIS
LIN {X 0.043,Y -407.656,Z 710.478,A 0.000,B 0.000,C 90.000,E1 85.988} C_DIS
LIN {X 0.105,Y -396.682,Z 710.467,A 0.000,B 0.000,C 90.000,E1 84.033} C_DIS
LIN {X 0.115,Y -379.725,Z 710.450,A 0.000,B 0.000,C 90.000,E1 80.905} C_DIS
LIN {X 0.120,Y -366.418,Z 710.435,A 0.000,B 0.000,C 90.000,E1 78.285} C_DIS
LIN {X -0.090,Y -353.648,Z 710.420,A 0.000,B 0.000,C 90.000,E1 75.644} C_DIS
LIN {X 0.053,Y -342.634,Z 710.407,A 0.000,B 0.000,C 90.000,E1 73.196} C_DIS
LIN {X 0.009,Y -330.634,Z 710.391,A 0.000,B 0.000,C 90.000,E1 70.423} C_DIS
LIN {X -0.080,Y -318.120,Z 710.374,A 0.000,B 0.000,C 90.000,E1 67.283} C_DIS
LIN {X -0.114,Y -309.248,Z 710.359,A 0.000,B 0.000,C 90.000,E1 64.717} C_DIS
LIN {X -0.032,Y -299.310,Z 710.341,A 0.000,B 0.000,C 90.000,E1 61.435} C_DIS
LIN {X -0.087,Y -290.022,Z 710.323,A 0.000,B 0.000,C 90.000,E1 58.122} C_DIS
LIN {X 0.176,Y -281.259,Z 710.304,A 0.000,B 0.000,C 90.000,E1 54.689} C_DIS
LIN {X -0.064,Y -276.121,Z 710.293,A 0.000,B 0.000,C 90.000,E1 52.683} C_DIS
LIN {X -0.012,Y -270.894,Z 710.281,A 0.000,B 0.000,C 90.000,E1 50.598} C_DIS
LIN {X 0.067,Y -265.464,Z 710.269,A 0.000,B 0.000,C 90.000,E1 48.485} C_DIS
LIN {X 0.024,Y -259.819,Z 710.258,A 0.000,B 0.000,C 90.000,E1 46.377} C_DIS
LIN {X -0.126,Y -253.968,Z 710.246,A 0.000,B 0.000,C 90.000,E1 44.271} C_DIS
LIN {X -0.017,Y -248.026,Z 710.234,A 0.000,B 0.000,C 90.000,E1 42.081} C_DIS
LIN {X 0.000,Y -241.917,Z 710.222,A 0.000,B 0.000,C 90.000,E1 39.886} C_DIS
LIN {X 0.017,Y -232.038,Z 710.201,A 0.000,B 0.000,C 90.000,E1 36.171} C_DIS
LIN {X -0.114,Y -222.960,Z 710.180,A 0.000,B 0.000,C 90.000,E1 32.418} C_DIS
LIN {X -0.089,Y -216.389,Z 710.163,A 0.000,B 0.000,C 90.000,E1 29.333} C_DIS
LIN {X 0.023,Y -210.632,Z 710.146,A 0.000,B 0.000,C 90.000,E1 26.181} C_DIS
LIN {X 0.003,Y -205.659,Z 710.128,A 0.000,B 0.000,C 90.000,E1 23.025} C_DIS
LIN {X -0.013,Y -200.515,Z 710.106,A 0.000,B 0.000,C 90.000,E1 19.033} C_DIS
LIN {X -0.069,Y -196.535,Z 710.083,A 0.000,B 0.000,C 90.000,E1 15.009} C_DIS
LIN {X 0.075,Y -193.186,Z 710.056,A 0.000,B 0.000,C 90.000,E1 10.074} C_DIS
LIN {X -0.041,Y -191.096,Z 710.010,A 0.000,B 0.000,C 90.000,E1 1.892} C_DIS
LIN {X -0.087,Y -193.073,Z 709.965,A 0.000,B 0.000,C 90.000,E1 353.799} C_DIS
LIN {X -0.032,Y -196.115,Z 709.938,A 0.000,B 0.000,C 90.000,E1 348.870} C_DIS
LIN {X -0.055,Y -199.799,Z 709.916,A 0.000,B 0.000,C 90.000,E1 344.810} C_DIS
LIN {X -0.080,Y -204.459,Z 709.893,A 0.000,B 0.000,C 90.000,E1 340.786} C_DIS
LIN {X -0.072,Y -209.963,Z 709.871,A 0.000,B 0.000,C 90.000,E1 336.794} C_DIS
LIN {X 0.050,Y -216.181,Z 709.849,A 0.000,B 0.000,C 90.000,E1 332.820} C_DIS
LIN {X -0.006,Y -223.094,Z 709.827,A 0.000,B 0.000,C 90.000,E1 328.948} C_DIS
LIN {X 0.057,Y -230.651,Z 709.806,A 0.000,B 0.000,C 90.000,E1 325.102} C_DIS
LIN {X 0.062,Y -238.791,Z 709.785,A 0.000,B 0.000,C 90.000,E1 321.331} C_DIS
LIN {X 0.025,Y -247.809,Z 709.765,A 0.000,B 0.000,C 90.000,E1 317.634} C_DIS
LIN {X -0.106,Y -257.908,Z 709.744,A 0.000,B 0.000,C 90.000,E1 314.028} C_DIS
LIN {X -0.058,Y -269.098,Z 709.725,A 0.000,B 0.000,C 90.000,E1 310.458} C_DIS
LIN {X -0.030,Y -280.292,Z 709.707,A 0.000,B 0.000,C 90.000,E1 307.317} C_DIS
LIN {X -0.035,Y -294.041,Z 709.688,A 0.000,B 0.000,C 90.000,E1 303.913} C_DIS
LIN {X -0.076,Y -306.061,Z 709.674,A 0.000,B 0.000,C 90.000,E1 301.258} C_DIS
LIN {X 0.139,Y -322.599,Z 709.656,A 0.000,B 0.000,C 90.000,E1 297.975} C_DIS
LIN {X 0.012,Y -340.732,Z 709.638,A 0.000,B 0.000,C 90.000,E1 294.847} C_DIS
LIN {X 0.081,Y -356.287,Z 709.624,A 0.000,B 0.000,C 90.000,E1 292.386} C_DIS
LIN {X 0.125,Y -372.600,Z 709.611,A 0.000,B 0.000,C 90.000,E1 289.993} C_DIS
LIN {X 0.185,Y -385.917,Z 709.601,A 0.000,B 0.000,C 90.000,E1 288.236} C_DIS
LIN {X -0.003,Y -399.941,Z 709.592,A 0.000,B 0.000,C 90.000,E1 286.551} C_DIS
LIN {X -0.169,Y -413.853,Z 709.583,A 0.000,B 0.000,C 90.000,E1 284.898} C_DIS
LIN {X -0.076,Y -427.470,Z 709.574,A 0.000,B 0.000,C 90.000,E1 283.244} C_DIS
LIN {X 0.059,Y -438.595,Z 709.566,A 0.000,B 0.000,C 90.000,E1 281.883} C_DIS
LIN {X 0.187,Y -448.942,Z 709.559,A 0.000,B 0.000,C 90.000,E1 280.546} C_DIS
LIN {X 0.044,Y -463.035,Z 709.549,A 0.000,B 0.000,C 90.000,E1 278.746} C_DIS
LIN {X 0.234,Y -470.864,Z 709.543,A 0.000,B 0.000,C 90.000,E1 277.701} C_DIS
LIN {X 0.185,Y -476.157,Z 709.539,A 0.000,B 0.000,C 90.000,E1 276.947} C_DIS
LIN {X 0.121,Y -480.711,Z 709.535,A 0.000,B 0.000,C 90.000,E1 276.201} C_DIS
LIN {X -0.199,Y -483.216,Z 709.532,A 0.000,B 0.000,C 90.000,E1 275.739} C_DIS
LIN {X -0.025,Y -485.298,Z 709.529,A 0.000,B 0.000,C 90.000,E1 275.220} C_DIS
LIN {X 0.162,Y -486.942,Z 709.526,A 0.000,B 0.000,C 90.000,E1 274.702} C_DIS
LIN {X -0.169,Y -488.156,Z 709.523,A 0.000,B 0.000,C 90.000,E1 274.245} C_DIS
LIN {X 0.033,Y -488.933,Z 709.521,A 0.000,B 0.000,C 90.000,E1 273.726} C_DIS
LIN {X 0.210,Y -489.361,Z 709.518,A 0.000,B 0.000,C 90.000,E1 273.212} C_DIS
LIN {X -0.069,Y -489.398,Z 709.515,A 0.000,B 0.000,C 90.000,E1 272.751} C_DIS
LIN {X 0.120,Y -489.100,Z 709.513,A 0.000,B 0.000,C 90.000,E1 272.236} C_DIS
LIN {X -0.163,Y -488.513,Z 709.510,A 0.000,B 0.000,C 90.000,E1 271.776} C_DIS
LIN {X 0.025,Y -487.520,Z 709.507,A 0.000,B 0.000,C 90.000,E1 271.260} C_DIS
LIN {X 0.209,Y -486.180,Z 709.504,A 0.000,B 0.000,C 90.000,E1 270.745} C_DIS
LIN {X -0.096,Y -484.357,Z 709.502,A 0.000,B 0.000,C 90.000,E1 270.286} C_DIS
LIN {X 0.076,Y -481.964,Z 709.499,A 0.000,B 0.000,C 90.000,E1 269.771} C_DIS
LIN {X 0.228,Y -478.910,Z 709.496,A 0.000,B 0.000,C 90.000,E1 269.255} C_DIS
LIN {X -0.112,Y -475.008,Z 709.493,A 0.000,B 0.000,C 90.000,E1 268.797} C_DIS
LIN {X 0.003,Y -470.148,Z 709.490,A 0.000,B 0.000,C 90.000,E1 268.282} C_DIS
LIN {X -0.219,Y -464.234,Z 709.488,A 0.000,B 0.000,C 90.000,E1 267.822} C_DIS
LIN {X -0.075,Y -461.164,Z 709.487,A 0.000,B 0.000,C 90.000,E1 267.593} C_DIS
LIN {X 0.054,Y -454.406,Z 709.484,A 0.000,B 0.000,C 90.000,E1 267.192} C_DIS
LIN {X 0.040,Y -450.761,Z 709.483,A 0.000,B 0.000,C 90.000,E1 267.020} C_DIS
LIN {X 0.074,Y -443.097,Z 709.482,A 0.000,B 0.000,C 90.000,E1 266.731} C_DIS
LIN {X 0.172,Y -435.036,Z 709.481,A 0.000,B 0.000,C 90.000,E1 266.502} C_DIS
LIN {X -0.129,Y -425.864,Z 709.480,A 0.000,B 0.000,C 90.000,E1 266.388} C_DIS
LIN {X -0.137,Y -415.880,Z 709.479,A 0.000,B 0.000,C 90.000,E1 266.331} C_DIS
LIN {X -0.081,Y -180.935,Z 709.479,A 0.000,B 0.000,C 90.000,E1 266.331} C_DIS
LIN {X -0.073,Y -180.717,Z 709.470,A 0.000,B 0.000,C 90.000,E1 264.609} C_DIS
LIN {X 0.026,Y -178.805,Z 709.442,A 0.000,B 0.000,C 90.000,E1 259.511} C_DIS
LIN {X -0.068,Y -175.850,Z 709.413,A 0.000,B 0.000,C 90.000,E1 254.448} C_DIS
LIN {X -0.101,Y -172.586,Z 709.390,A 0.000,B 0.000,C 90.000,E1 250.188} C_DIS
LIN {X 0.076,Y -171.476,Z 709.380,A 0.000,B 0.000,C 90.000,E1 248.411} C_DIS
LIN {X -0.095,Y -167.706,Z 709.356,A 0.000,B 0.000,C 90.000,E1 244.152} C_DIS
LIN {X 0.070,Y -166.394,Z 709.347,A 0.000,B 0.000,C 90.000,E1 242.359} C_DIS
LIN {X 0.061,Y -163.120,Z 709.327,A 0.000,B 0.000,C 90.000,E1 238.869} C_DIS
LIN {X 0.021,Y -161.070,Z 709.313,A 0.000,B 0.000,C 90.000,E1 236.246} C_DIS
LIN {X -0.003,Y -157.803,Z 709.293,A 0.000,B 0.000,C 90.000,E1 232.718} C_DIS
LIN {X -0.064,Y -155.839,Z 709.278,A 0.000,B 0.000,C 90.000,E1 230.070} C_DIS
LIN {X -0.007,Y -152.088,Z 709.253,A 0.000,B 0.000,C 90.000,E1 225.567} C_DIS
LIN {X 0.011,Y -150.339,Z 709.238,A 0.000,B 0.000,C 90.000,E1 222.852} C_DIS
LIN {X 0.032,Y -147.078,Z 709.213,A 0.000,B 0.000,C 90.000,E1 218.302} C_DIS
LIN {X -0.064,Y -145.651,Z 709.198,A 0.000,B 0.000,C 90.000,E1 215.598} C_DIS
LIN {X -0.060,Y -143.034,Z 709.172,A 0.000,B 0.000,C 90.000,E1 211.003} C_DIS
LIN {X 0.066,Y -141.659,Z 709.152,A 0.000,B 0.000,C 90.000,E1 207.257} C_DIS
LIN {X -0.015,Y -139.447,Z 709.115,A 0.000,B 0.000,C 90.000,E1 200.791} C_DIS
LIN {X 0.038,Y -139.180,Z 709.105,A 0.000,B 0.000,C 90.000,E1 198.906} C_DIS
LIN {X 0.066,Y -138.321,Z 709.053,A 0.000,B 0.000,C 90.000,E1 189.557} C_DIS
LIN {X -0.063,Y -139.465,Z 709.007,A 0.000,B 0.000,C 90.000,E1 181.203} C_DIS
LIN {X 0.017,Y -141.028,Z 708.976,A 0.000,B 0.000,C 90.000,E1 175.584} C_DIS
LIN {X -0.029,Y -142.394,Z 708.960,A 0.000,B 0.000,C 90.000,E1 172.818} C_DIS
LIN {X 0.034,Y -144.625,Z 708.934,A 0.000,B 0.000,C 90.000,E1 168.173} C_DIS
LIN {X -0.047,Y -147.821,Z 708.909,A 0.000,B 0.000,C 90.000,E1 163.614} C_DIS
LIN {X 0.039,Y -150.512,Z 708.889,A 0.000,B 0.000,C 90.000,E1 159.934} C_DIS
LIN {X 0.059,Y -153.972,Z 708.868,A 0.000,B 0.000,C 90.000,E1 156.305} C_DIS
LIN {X -0.019,Y -157.384,Z 708.849,A 0.000,B 0.000,C 90.000,E1 152.743} C_DIS
LIN {X -0.077,Y -161.587,Z 708.829,A 0.000,B 0.000,C 90.000,E1 149.203} C_DIS
LIN {X -0.067,Y -165.784,Z 708.809,A 0.000,B 0.000,C 90.000,E1 145.674} C_DIS
LIN {X -0.081,Y -170.746,Z 708.790,A 0.000,B 0.000,C 90.000,E1 142.190} C_DIS
LIN {X 0.077,Y -175.618,Z 708.771,A 0.000,B 0.000,C 90.000,E1 138.690} C_DIS
LIN {X -0.054,Y -181.234,Z 708.752,A 0.000,B 0.000,C 90.000,E1 135.324} C_DIS
LIN {X 0.077,Y -186.703,Z 708.733,A 0.000,B 0.000,C 90.000,E1 131.919} C_DIS
LIN {X 0.062,Y -191.418,Z 708.719,A 0.000,B 0.000,C 90.000,E1 129.358} C_DIS
LIN {X 0.059,Y -289.264,Z 708.719,A 0.000,B 0.000,C 90.000,E1 129.358} C_DIS
LIN {X 0.154,Y -292.555,Z 708.718,A 0.000,B 0.000,C 90.000,E1 129.277} C_DIS
LIN {X 0.048,Y -297.946,Z 708.716,A 0.000,B 0.000,C 90.000,E1 128.955} C_DIS
LIN {X -0.015,Y -300.904,Z 708.715,A 0.000,B 0.000,C 90.000,E1 128.624} C_DIS
LIN {X 0.011,Y -302.894,Z 708.713,A 0.000,B 0.000,C 90.000,E1 128.302} C_DIS
LIN {X 0.086,Y -304.447,Z 708.711,A 0.000,B 0.000,C 90.000,E1 127.971} C_DIS
LIN {X 0.047,Y -305.720,Z 708.709,A 0.000,B 0.000,C 90.000,E1 127.649} C_DIS
LIN {X -0.201,Y -317.453,Z 708.688,A 0.000,B 0.000,C 90.000,E1 123.785} C_DIS
LIN {X 0.004,Y -327.603,Z 708.672,A 0.000,B 0.000,C 90.000,E1 120.875} C_DIS
LIN {X 0.015,Y -339.084,Z 708.656,A 0.000,B 0.000,C 90.000,E1 118.052} C_DIS
LIN {X 0.035,Y -352.006,Z 708.641,A 0.000,B 0.000,C 90.000,E1 115.283} C_DIS
LIN {X -0.101,Y -364.791,Z 708.627,A 0.000,B 0.000,C 90.000,E1 112.898} C_DIS
LIN {X -0.072,Y -378.894,Z 708.614,A 0.000,B 0.000,C 90.000,E1 110.536} C_DIS
LIN {X -0.095,Y -394.416,Z 708.601,A 0.000,B 0.000,C 90.000,E1 108.236} C_DIS
LIN {X 0.041,Y -411.471,Z 708.589,A 0.000,B 0.000,C 90.000,E1 105.969} C_DIS
LIN {X 0.105,Y -430.182,Z 708.577,A 0.000,B 0.000,C 90.000,E1 103.772} C_DIS
LIN {X -0.045,Y -450.173,Z 708.565,A 0.000,B 0.000,C 90.000,E1 101.715} C_DIS
LIN {X 0.134,Y -468.109,Z 708.556,A 0.000,B 0.000,C 90.000,E1 100.018} C_DIS
LIN {X 0.096,Y -470.262,Z 708.554,A 0.000,B 0.000,C 90.000,E1 99.792} C_DIS
LIN {X -0.054,Y -472.037,Z 708.553,A 0.000,B 0.000,C 90.000,E1 99.557} C_DIS
LIN {X -0.206,Y -473.370,Z 708.552,A 0.000,B 0.000,C 90.000,E1 99.321} C_DIS
LIN {X -0.096,Y -475.038,Z 708.549,A 0.000,B 0.000,C 90.000,E1 98.803} C_DIS
LIN {X 0.095,Y -475.639,Z 708.546,A 0.000,B 0.000,C 90.000,E1 98.276} C_DIS
LIN {X 0.224,Y -475.275,Z 708.543,A 0.000,B 0.000,C 90.000,E1 97.757} C_DIS
LIN {X -0.112,Y -473.892,Z 708.540,A 0.000,B 0.000,C 90.000,E1 97.296} C_DIS
LIN {X 0.160,Y -472.751,Z 708.539,A 0.000,B 0.000,C 90.000,E1 97.011} C_DIS
LIN {X 0.138,Y -467.838,Z 708.535,A 0.000,B 0.000,C 90.000,E1 96.258} C_DIS
LIN {X -0.067,Y -451.706,Z 708.521,A 0.000,B 0.000,C 90.000,E1 93.726} C_DIS
LIN {X -0.055,Y -438.452,Z 708.508,A 0.000,B 0.000,C 90.000,E1 91.375} C_DIS
LIN {X 0.038,Y -429.459,Z 708.499,A 0.000,B 0.000,C 90.000,E1 89.771} C_DIS
LIN {X -0.016,Y -420.165,Z 708.490,A 0.000,B 0.000,C 90.000,E1 88.165} C_DIS
LIN {X -0.071,Y -407.640,Z 708.478,A 0.000,B 0.000,C 90.000,E1 85.988} C_DIS
LIN {X -0.044,Y -398.233,Z 708.468,A 0.000,B 0.000,C 90.000,E1 84.318} C_DIS
LIN {X -0.090,Y -384.258,Z 708.454,A 0.000,B 0.000,C 90.000,E1 81.781} C_DIS
LIN {X 0.031,Y -370.832,Z 708.440,A 0.000,B 0.000,C 90.000,E1 79.162} C_DIS
LIN {X -0.095,Y -356.500,Z 708.423,A 0.000,B 0.000,C 90.000,E1 76.228} C_DIS
LIN {X -0.051,Y -344.091,Z 708.408,A 0.000,B 0.000,C 90.000,E1 73.504} C_DIS
LIN {X -0.062,Y -332.072,Z 708.393,A 0.000,B 0.000,C 90.000,E1 70.732} C_DIS
LIN {X 0.133,Y -318.275,Z 708.374,A 0.000,B 0.000,C 90.000,E1 67.230} C_DIS
LIN {X 0.098,Y -309.436,Z 708.359,A 0.000,B 0.000,C 90.000,E1 64.665} C_DIS
LIN {X -0.091,Y -299.520,Z 708.341,A 0.000,B 0.000,C 90.000,E1 61.435} C_DIS
LIN {X 0.108,Y -290.259,Z 708.323,A 0.000,B 0.000,C 90.000,E1 58.074} C_DIS
LIN {X 0.040,Y -283.223,Z 708.308,A 0.000,B 0.000,C 90.000,E1 55.388} C_DIS
LIN {X 0.120,Y -276.397,Z 708.293,A 0.000,B 0.000,C 90.000,E1 52.637} C_DIS
LIN {X -0.043,Y -271.184,Z 708.281,A 0.000,B 0.000,C 90.000,E1 50.598} C_DIS
LIN {X 0.042,Y -265.762,Z 708.269,A 0.000,B 0.000,C 90.000,E1 48.485} C_DIS
LIN {X 0.005,Y -260.106,Z 708.258,A 0.000,B 0.000,C 90.000,E1 46.377} C_DIS
LIN {X -0.140,Y -254.238,Z 708.246,A 0.000,B 0.000,C 90.000,E1 44.271} C_DIS
LIN {X -0.025,Y -248.310,Z 708.234,A 0.000,B 0.000,C 90.000,E1 42.081} C_DIS
LIN {X -0.003,Y -242.148,Z 708.222,A 0.000,B 0.000,C 90.000,E1 39.886} C_DIS
LIN {X 0.022,Y -232.252,Z 708.201,A 0.000,B 0.000,C 90.000,E1 36.171} C_DIS
LIN {X -0.104,Y -223.142,Z 708.180,A 0.000,B 0.000,C 90.000,E1 32.418} C_DIS
LIN {X -0.075,Y -216.559,Z 708.163,A 0.000,B 0.000,C 90.000,E1 29.333} C_DIS
LIN {X 0.042,Y -210.790,Z 708.146,A 0.000,B 0.000,C 90.000,E1 26.181} C_DIS
LIN {X 0.025,Y -205.789,Z 708.128,A 0.000,B 0.000,C 90.000,E1 23.025} C_DIS
LIN {X 0.012,Y -200.650,Z 708.106,A 0.000,B 0.000,C 90.000,E1 19.033} C_DIS
LIN {X -0.041,Y -196.680,Z 708.083,A 0.000,B 0.000,C 90.000,E1 15.009} C_DIS
LIN {X 0.075,Y -193.333,Z 708.056,A 0.000,B 0.000,C 90.000,E1 10.084} C_DIS
LIN {X 0.001,Y -191.230,Z 708.010,A 0.000,B 0.000,C 90.000,E1 1.892} C_DIS
LIN {X -0.082,Y -193.195,Z 707.965,A 0.000,B 0.000,C 90.000,E1 353.799} C_DIS
LIN {X -0.023,Y -196.228,Z 707.938,A 0.000,B 0.000,C 90.000,E1 348.870} C_DIS
LIN {X -0.042,Y -199.902,Z 707.916,A 0.000,B 0.000,C 90.000,E1 344.810} C_DIS
LIN {X -0.064,Y -204.548,Z 707.893,A 0.000,B 0.000,C 90.000,E1 340.786} C_DIS
LIN {X -0.053,Y -210.036,Z 707.871,A 0.000,B 0.000,C 90.000,E1 336.794} C_DIS
LIN {X -0.119,Y -216.245,Z 707.849,A 0.000,B 0.000,C 90.000,E1 332.871} C_DIS
LIN {X 0.019,Y -223.145,Z 707.828,A 0.000,B 0.000,C 90.000,E1 328.948} C_DIS
LIN {X 0.085,Y -230.689,Z 707.806,A 0.000,B 0.000,C 90.000,E1 325.102} C_DIS
LIN {X 0.092,Y -238.802,Z 707.785,A 0.000,B 0.000,C 90.000,E1 321.331} C_DIS
LIN {X 0.056,Y -247.829,Z 707.765,A 0.000,B 0.000,C 90.000,E1 317.634} C_DIS
LIN {X -0.073,Y -257.923,Z 707.745,A 0.000,B 0.000,C 90.000,E1 314.028} C_DIS
LIN {X -0.023,Y -269.122,Z 707.725,A 0.000,B 0.000,C 90.000,E1 310.458} C_DIS
LIN {X 0.007,Y -280.308,Z 707.707,A 0.000,B 0.000,C 90.000,E1 307.317} C_DIS
LIN {X 0.005,Y -294.065,Z 707.688,A 0.000,B 0.000,C 90.000,E1 303.913} C_DIS
LIN {X -0.007,Y -307.666,Z 707.672,A 0.000,B 0.000,C 90.000,E1 300.924} C_DIS
LIN {X -0.175,Y -324.337,Z 707.654,A 0.000,B 0.000,C 90.000,E1 297.719} C_DIS
LIN {X 0.060,Y -340.697,Z 707.638,A 0.000,B 0.000,C 90.000,E1 294.847} C_DIS
LIN {X -0.006,Y -356.222,Z 707.625,A 0.000,B 0.000,C 90.000,E1 292.408} C_DIS
LIN {X 0.174,Y -372.459,Z 707.611,A 0.000,B 0.000,C 90.000,E1 289.993} C_DIS
LIN {X -0.125,Y -388.091,Z 707.600,A 0.000,B 0.000,C 90.000,E1 288.000} C_DIS
LIN {X 0.103,Y -402.131,Z 707.590,A 0.000,B 0.000,C 90.000,E1 286.260} C_DIS
LIN {X 0.092,Y -415.971,Z 707.581,A 0.000,B 0.000,C 90.000,E1 284.592} C_DIS
LIN {X -0.033,Y -427.312,Z 707.574,A 0.000,B 0.000,C 90.000,E1 283.244} C_DIS
LIN {X -0.088,Y -436.237,Z 707.568,A 0.000,B 0.000,C 90.000,E1 282.175} C_DIS
LIN {X -0.227,Y -444.636,Z 707.562,A 0.000,B 0.000,C 90.000,E1 281.130} C_DIS
LIN {X -0.201,Y -456.747,Z 707.553,A 0.000,B 0.000,C 90.000,E1 279.557} C_DIS
LIN {X 0.195,Y -466.757,Z 707.546,A 0.000,B 0.000,C 90.000,E1 278.219} C_DIS
LIN {X 0.050,Y -472.498,Z 707.542,A 0.000,B 0.000,C 90.000,E1 277.473} C_DIS
LIN {X 0.012,Y -477.579,Z 707.537,A 0.000,B 0.000,C 90.000,E1 276.720} C_DIS
LIN {X 0.152,Y -480.548,Z 707.535,A 0.000,B 0.000,C 90.000,E1 276.201} C_DIS
LIN {X 0.136,Y -484.165,Z 707.530,A 0.000,B 0.000,C 90.000,E1 275.454} C_DIS
LIN {X 0.190,Y -486.793,Z 707.526,A 0.000,B 0.000,C 90.000,E1 274.702} C_DIS
LIN {X -0.141,Y -488.029,Z 707.523,A 0.000,B 0.000,C 90.000,E1 274.245} C_DIS
LIN {X 0.060,Y -488.832,Z 707.521,A 0.000,B 0.000,C 90.000,E1 273.726} C_DIS
LIN {X -0.252,Y -489.277,Z 707.518,A 0.000,B 0.000,C 90.000,E1 273.269} C_DIS
LIN {X -0.043,Y -489.323,Z 707.515,A 0.000,B 0.000,C 90.000,E1 272.751} C_DIS
LIN {X 0.145,Y -489.044,Z 707.513,A 0.000,B 0.000,C 90.000,E1 272.236} C_DIS
LIN {X -0.138,Y -488.443,Z 707.510,A 0.000,B 0.000,C 90.000,E1 271.776} C_DIS
LIN {X 0.049,Y -487.472,Z 707.507,A 0.000,B 0.000,C 90.000,E1 271.260} C_DIS
LIN {X 0.233,Y -486.092,Z 707.504,A 0.000,B 0.000,C 90.000,E1 270.745} C_DIS
LIN {X -0.072,Y -484.276,Z 707.502,A 0.000,B 0.000,C 90.000,E1 270.286} C_DIS
LIN {X 0.098,Y -481.878,Z 707.499,A 0.000,B 0.000,C 90.000,E1 269.771} C_DIS
LIN {X -0.228,Y -478.854,Z 707.496,A 0.000,B 0.000,C 90.000,E1 269.312} C_DIS
LIN {X -0.090,Y -474.977,Z 707.493,A 0.000,B 0.000,C 90.000,E1 268.797} C_DIS
LIN {X 0.024,Y -470.107,Z 707.490,A 0.000,B 0.000,C 90.000,E1 268.282} C_DIS
LIN {X -0.075,Y -467.369,Z 707.489,A 0.000,B 0.000,C 90.000,E1 268.051} C_DIS
LIN {X -0.021,Y -461.230,Z 707.487,A 0.000,B 0.000,C 90.000,E1 267.593} C_DIS
LIN {X 0.118,Y -454.579,Z 707.484,A 0.000,B 0.000,C 90.000,E1 267.192} C_DIS
LIN {X 0.094,Y -450.926,Z 707.484,A 0.000,B 0.000,C 90.000,E1 267.020} C_DIS
LIN {X 0.116,Y -443.337,Z 707.482,A 0.000,B 0.000,C 90.000,E1 266.731} C_DIS
LIN {X 0.197,Y -435.437,Z 707.481,A 0.000,B 0.000,C 90.000,E1 266.502} C_DIS
LIN {X -0.151,Y -426.178,Z 707.480,A 0.000,B 0.000,C 90.000,E1 266.388} C_DIS
LIN {X -0.163,Y -416.671,Z 707.479,A 0.000,B 0.000,C 90.000,E1 266.331} C_DIS
LIN {X 0.088,Y -180.935,Z 707.479,A 0.000,B 0.000,C 90.000,E1 266.274} C_DIS
LIN {X -0.090,Y -180.715,Z 707.470,A 0.000,B 0.000,C 90.000,E1 264.609} C_DIS
LIN {X 0.008,Y -178.802,Z 707.442,A 0.000,B 0.000,C 90.000,E1 259.511} C_DIS
LIN {X 0.085,Y -175.848,Z 707.413,A 0.000,B 0.000,C 90.000,E1 254.393} C_DIS
LIN {X 0.044,Y -172.582,Z 707.390,A 0.000,B 0.000,C 90.000,E1 250.134} C_DIS
LIN {X 0.059,Y -171.471,Z 707.380,A 0.000,B 0.000,C 90.000,E1 248.411} C_DIS
LIN {X 0.039,Y -167.702,Z 707.356,A 0.000,B 0.000,C 90.000,E1 244.101} C_DIS
LIN {X 0.053,Y -166.388,Z 707.347,A 0.000,B 0.000,C 90.000,E1 242.359} C_DIS
LIN {X 0.044,Y -163.116,Z 707.327,A 0.000,B 0.000,C 90.000,E1 238.869} C_DIS
LIN {X 0.094,Y -161.064,Z 707.313,A 0.000,B 0.000,C 90.000,E1 236.215} C_DIS
LIN {X -0.019,Y -157.798,Z 707.293,A 0.000,B 0.000,C 90.000,E1 232.718} C_DIS
LIN {X 0.020,Y -155.834,Z 707.278,A 0.000,B 0.000,C 90.000,E1 230.033} C_DIS
LIN {X -0.024,Y -152.085,Z 707.253,A 0.000,B 0.000,C 90.000,E1 225.567} C_DIS
LIN {X -0.005,Y -150.335,Z 707.238,A 0.000,B 0.000,C 90.000,E1 222.852} C_DIS
LIN {X 0.017,Y -147.075,Z 707.213,A 0.000,B 0.000,C 90.000,E1 218.302} C_DIS
LIN {X -0.080,Y -145.649,Z 707.198,A 0.000,B 0.000,C 90.000,E1 215.598} C_DIS
LIN {X -0.075,Y -143.030,Z 707.172,A 0.000,B 0.000,C 90.000,E1 211.003} C_DIS
LIN {X 0.052,Y -141.656,Z 707.152,A 0.000,B 0.000,C 90.000,E1 207.257} C_DIS
LIN {X -0.029,Y -139.446,Z 707.115,A 0.000,B 0.000,C 90.000,E1 200.791} C_DIS
LIN {X 0.023,Y -139.179,Z 707.105,A 0.000,B 0.000,C 90.000,E1 198.906} C_DIS
LIN {X 0.052,Y -138.320,Z 707.053,A 0.000,B 0.000,C 90.000,E1 189.557} C_DIS
LIN {X 0.061,Y -139.466,Z 707.007,A 0.000,B 0.000,C 90.000,E1 181.146} C_DIS
LIN {X 0.002,Y -141.031,Z 706.975,A 0.000,B 0.000,C 90.000,E1 175.584} C_DIS
LIN {X -0.044,Y -142.397,Z 706.960,A 0.000,B 0.000,C 90.000,E1 172.818} C_DIS
LIN {X 0.019,Y -144.629,Z 706.934,A 0.000,B 0.000,C 90.000,E1 168.173} C_DIS
LIN {X 0.079,Y -147.824,Z 706.909,A 0.000,B 0.000,C 90.000,E1 163.559} C_DIS
LIN {X 0.024,Y -150.517,Z 706.889,A 0.000,B 0.000,C 90.000,E1 159.934} C_DIS
LIN {X 0.043,Y -153.978,Z 706.868,A 0.000,B 0.000,C 90.000,E1 156.305} C_DIS
LIN {X -0.036,Y -157.391,Z 706.849,A 0.000,B 0.000,C 90.000,E1 152.743} C_DIS
LIN {X -0.093,Y -161.595,Z 706.829,A 0.000,B 0.000,C 90.000,E1 149.203} C_DIS
LIN {X -0.083,Y -165.792,Z 706.809,A 0.000,B 0.000,C 90.000,E1 145.674} C_DIS
LIN {X -0.098,Y -170.755,Z 706.790,A 0.000,B 0.000,C 90.000,E1 142.190} C_DIS
LIN {X 0.059,Y -175.626,Z 706.771,A 0.000,B 0.000,C 90.000,E1 138.690} C_DIS
LIN {X -0.071,Y -181.242,Z 706.752,A 0.000,B 0.000,C 90.000,E1 135.324} C_DIS
LIN {X 0.059,Y -186.712,Z 706.733,A 0.000,B 0.000,C 90.000,E1 131.919} C_DIS
LIN {X -0.033,Y -191.392,Z 706.719,A 0.000,B 0.000,C 90.000,E1 129.402} C_DIS
LIN {X 0.121,Y -289.319,Z 706.719,A 0.000,B 0.000,C 90.000,E1 129.358} C_DIS
LIN {X 0.067,Y -290.445,Z 706.719,A 0.000,B 0.000,C 90.000,E1 129.358} C_DIS
LIN {X -0.074,Y -295.289,Z 706.718,A 0.000,B 0.000,C 90.000,E1 129.197} C_DIS
LIN {X 0.013,Y -297.715,Z 706.717,A 0.000,B 0.000,C 90.000,E1 128.991} C_DIS
LIN {X -0.043,Y -300.980,Z 706.715,A 0.000,B 0.000,C 90.000,E1 128.624} C_DIS
LIN {X -0.015,Y -302.936,Z 706.713,A 0.000,B 0.000,C 90.000,E1 128.302} C_DIS
LIN {X 0.064,Y -304.466,Z 706.711,A 0.000,B 0.000,C 90.000,E1 127.971} C_DIS
LIN {X 0.024,Y -305.724,Z 706.709,A 0.000,B 0.000,C 90.000,E1 127.649} C_DIS
LIN {X 0.216,Y -317.447,Z 706.688,A 0.000,B 0.000,C 90.000,E1 123.706} C_DIS
LIN {X -0.021,Y -327.598,Z 706.672,A 0.000,B 0.000,C 90.000,E1 120.875} C_DIS
LIN {X 0.149,Y -339.082,Z 706.656,A 0.000,B 0.000,C 90.000,E1 118.025} C_DIS
LIN {X 0.008,Y -352.006,Z 706.640,A 0.000,B 0.000,C 90.000,E1 115.283} C_DIS
LIN {X -0.128,Y -364.792,Z 706.627,A 0.000,B 0.000,C 90.000,E1 112.898} C_DIS
LIN {X -0.100,Y -378.897,Z 706.614,A 0.000,B 0.000,C 90.000,E1 110.536} C_DIS
LIN {X -0.125,Y -394.422,Z 706.601,A 0.000,B 0.000,C 90.000,E1 108.236} C_DIS
LIN {X 0.010,Y -411.479,Z 706.589,A 0.000,B 0.000,C 90.000,E1 105.969} C_DIS
LIN {X 0.073,Y -430.193,Z 706.577,A 0.000,B 0.000,C 90.000,E1 103.772} C_DIS
LIN {X -0.077,Y -450.186,Z 706.565,A 0.000,B 0.000,C 90.000,E1 101.715} C_DIS
LIN {X 0.102,Y -468.124,Z 706.556,A 0.000,B 0.000,C 90.000,E1 100.018} C_DIS
LIN {X 0.065,Y -470.284,Z 706.554,A 0.000,B 0.000,C 90.000,E1 99.792} C_DIS
LIN {X -0.085,Y -472.066,Z 706.553,A 0.000,B 0.000,C 90.000,E1 99.557} C_DIS
LIN {X 0.230,Y -473.403,Z 706.552,A 0.000,B 0.000,C 90.000,E1 99.265} C_DIS
LIN {X -0.128,Y -475.077,Z 706.549,A 0.000,B 0.000,C 90.000,E1 98.803} C_DIS
LIN {X 0.063,Y -475.685,Z 706.546,A 0.000,B 0.000,C 90.000,E1 98.276} C_DIS
LIN {X 0.193,Y -475.326,Z 706.543,A 0.000,B 0.000,C 90.000,E1 97.757} C_DIS
LIN {X -0.143,Y -473.951,Z 706.540,A 0.000,B 0.000,C 90.000,E1 97.296} C_DIS
LIN {X 0.129,Y -472.812,Z 706.539,A 0.000,B 0.000,C 90.000,E1 97.011} C_DIS
LIN {X -0.156,Y -469.588,Z 706.536,A 0.000,B 0.000,C 90.000,E1 96.543} C_DIS
LIN {X -0.093,Y -451.744,Z 706.521,A 0.000,B 0.000,C 90.000,E1 93.726} C_DIS
LIN {X 0.094,Y -437.043,Z 706.506,A 0.000,B 0.000,C 90.000,E1 91.088} C_DIS
LIN {X 0.160,Y -427.983,Z 706.497,A 0.000,B 0.000,C 90.000,E1 89.484} C_DIS
LIN {X 0.077,Y -418.660,Z 706.488,A 0.000,B 0.000,C 90.000,E1 87.879} C_DIS
LIN {X -0.091,Y -407.699,Z 706.478,A 0.000,B 0.000,C 90.000,E1 85.988} C_DIS
LIN {X -0.063,Y -398.313,Z 706.468,A 0.000,B 0.000,C 90.000,E1 84.318} C_DIS
LIN {X -0.071,Y -382.836,Z 706.453,A 0.000,B 0.000,C 90.000,E1 81.489} C_DIS
LIN {X 0.020,Y -369.480,Z 706.438,A 0.000,B 0.000,C 90.000,E1 78.870} C_DIS
LIN {X -0.146,Y -355.236,Z 706.422,A 0.000,B 0.000,C 90.000,E1 75.936} C_DIS
LIN {X -0.135,Y -341.521,Z 706.405,A 0.000,B 0.000,C 90.000,E1 72.906} C_DIS
LIN {X -0.080,Y -330.955,Z 706.391,A 0.000,B 0.000,C 90.000,E1 70.423} C_DIS
LIN {X 0.139,Y -318.493,Z 706.374,A 0.000,B 0.000,C 90.000,E1 67.230} C_DIS
LIN {X 0.109,Y -309.672,Z 706.359,A 0.000,B 0.000,C 90.000,E1 64.665} C_DIS
LIN {X -0.074,Y -299.772,Z 706.341,A 0.000,B 0.000,C 90.000,E1 61.435} C_DIS
LIN {X -0.113,Y -290.536,Z 706.323,A 0.000,B 0.000,C 90.000,E1 58.122} C_DIS
LIN {X 0.070,Y -283.527,Z 706.308,A 0.000,B 0.000,C 90.000,E1 55.388} C_DIS
LIN {X -0.062,Y -276.725,Z 706.293,A 0.000,B 0.000,C 90.000,E1 52.683} C_DIS
LIN {X 0.000,Y -271.497,Z 706.281,A 0.000,B 0.000,C 90.000,E1 50.598} C_DIS
LIN {X 0.091,Y -266.109,Z 706.269,A 0.000,B 0.000,C 90.000,E1 48.485} C_DIS
LIN {X 0.058,Y -260.423,Z 706.258,A 0.000,B 0.000,C 90.000,E1 46.377} C_DIS
LIN {X -0.081,Y -254.598,Z 706.246,A 0.000,B 0.000,C 90.000,E1 44.271} C_DIS
LIN {X 0.038,Y -248.599,Z 706.234,A 0.000,B 0.000,C 90.000,E1 42.081} C_DIS
LIN {X 0.064,Y -242.434,Z 706.222,A 0.000,B 0.000,C 90.000,E1 39.886} C_DIS
LIN {X -0.093,Y -232.505,Z 706.201,A 0.000,B 0.000,C 90.000,E1 36.217} C_DIS
LIN {X -0.026,Y -223.358,Z 706.180,A 0.000,B 0.000,C 90.000,E1 32.418} C_DIS
LIN {X 0.005,Y -216.756,Z 706.163,A 0.000,B 0.000,C 90.000,E1 29.333} C_DIS
LIN {X -0.065,Y -210.978,Z 706.146,A 0.000,B 0.000,C 90.000,E1 26.232} C_DIS
LIN {X -0.080,Y -205.943,Z 706.128,A 0.000,B 0.000,C 90.000,E1 23.078} C_DIS
LIN {X -0.090,Y -200.806,Z 706.106,A 0.000,B 0.000,C 90.000,E1 19.087} C_DIS
LIN {X 0.052,Y -196.843,Z 706.083,A 0.000,B 0.000,C 90.000,E1 15.009} C_DIS
LIN {X -0.020,Y -193.491,Z 706.056,A 0.000,B 0.000,C 90.000,E1 10.141} C_DIS
LIN {X -0.086,Y -191.366,Z 706.011,A 0.000,B 0.000,C 90.000,E1 1.949} C_DIS
LIN {X -0.077,Y -193.318,Z 705.965,A 0.000,B 0.000,C 90.000,E1 353.799} C_DIS
LIN {X -0.013,Y -196.342,Z 705.938,A 0.000,B 0.000,C 90.000,E1 348.870} C_DIS
LIN {X -0.028,Y -200.009,Z 705.916,A 0.000,B 0.000,C 90.000,E1 344.810} C_DIS
LIN {X -0.046,Y -204.636,Z 705.893,A 0.000,B 0.000,C 90.000,E1 340.786} C_DIS
LIN {X -0.032,Y -210.108,Z 705.871,A 0.000,B 0.000,C 90.000,E1 336.794} C_DIS
LIN {X -0.096,Y -216.300,Z 705.849,A 0.000,B 0.000,C 90.000,E1 332.871} C_DIS
LIN {X 0.044,Y -223.193,Z 705.828,A 0.000,B 0.000,C 90.000,E1 328.948} C_DIS
LIN {X 0.112,Y -230.716,Z 705.806,A 0.000,B 0.000,C 90.000,E1 325.102} C_DIS
LIN {X -0.064,Y -238.829,Z 705.785,A 0.000,B 0.000,C 90.000,E1 321.376} C_DIS
LIN {X 0.088,Y -247.849,Z 705.765,A 0.000,B 0.000,C 90.000,E1 317.634} C_DIS
LIN {X -0.039,Y -257.938,Z 705.745,A 0.000,B 0.000,C 90.000,E1 314.028} C_DIS
LIN {X 0.013,Y -269.139,Z 705.725,A 0.000,B 0.000,C 90.000,E1 310.458} C_DIS
LIN {X 0.045,Y -280.319,Z 705.707,A 0.000,B 0.000,C 90.000,E1 307.317} C_DIS
LIN {X 0.046,Y -294.089,Z 705.688,A 0.000,B 0.000,C 90.000,E1 303.913} C_DIS
LIN {X 0.073,Y -309.271,Z 705.670,A 0.000,B 0.000,C 90.000,E1 300.590} C_DIS
LIN {X -0.130,Y -324.330,Z 705.654,A 0.000,B 0.000,C 90.000,E1 297.719} C_DIS
LIN {X -0.072,Y -342.572,Z 705.636,A 0.000,B 0.000,C 90.000,E1 294.567} C_DIS
LIN {X 0.082,Y -358.118,Z 705.623,A 0.000,B 0.000,C 90.000,E1 292.099} C_DIS
LIN {X 0.222,Y -372.316,Z 705.611,A 0.000,B 0.000,C 90.000,E1 289.993} C_DIS
LIN {X 0.067,Y -390.271,Z 705.598,A 0.000,B 0.000,C 90.000,E1 287.692} C_DIS
LIN {X 0.151,Y -401.959,Z 705.590,A 0.000,B 0.000,C 90.000,E1 286.260} C_DIS
LIN {X 0.137,Y -415.787,Z 705.581,A 0.000,B 0.000,C 90.000,E1 284.592} C_DIS
LIN {X 0.011,Y -427.145,Z 705.574,A 0.000,B 0.000,C 90.000,E1 283.244} C_DIS
LIN {X -0.045,Y -436.020,Z 705.568,A 0.000,B 0.000,C 90.000,E1 282.175} C_DIS
LIN {X -0.186,Y -444.413,Z 705.562,A 0.000,B 0.000,C 90.000,E1 281.130} C_DIS
LIN {X 0.096,Y -458.513,Z 705.552,A 0.000,B 0.000,C 90.000,E1 279.265} C_DIS
LIN {X 0.001,Y -468.514,Z 705.544,A 0.000,B 0.000,C 90.000,E1 277.992} C_DIS
LIN {X -0.073,Y -474.058,Z 705.540,A 0.000,B 0.000,C 90.000,E1 277.239} C_DIS
LIN {X -0.098,Y -478.939,Z 705.536,A 0.000,B 0.000,C 90.000,E1 276.486} C_DIS
LIN {X 0.048,Y -481.702,Z 705.533,A 0.000,B 0.000,C 90.000,E1 275.967} C_DIS
LIN {X 0.165,Y -484.006,Z 705.530,A 0.000,B 0.000,C 90.000,E1 275.454} C_DIS
LIN {X 0.034,Y -485.016,Z 705.529,A 0.000,B 0.000,C 90.000,E1 275.220} C_DIS
LIN {X 0.219,Y -486.676,Z 705.526,A 0.000,B 0.000,C 90.000,E1 274.702} C_DIS
LIN {X -0.113,Y -487.908,Z 705.523,A 0.000,B 0.000,C 90.000,E1 274.245} C_DIS
LIN {X 0.087,Y -488.737,Z 705.521,A 0.000,B 0.000,C 90.000,E1 273.726} C_DIS
LIN {X -0.225,Y -489.148,Z 705.518,A 0.000,B 0.000,C 90.000,E1 273.269} C_DIS
LIN {X -0.017,Y -489.233,Z 705.515,A 0.000,B 0.000,C 90.000,E1 272.751} C_DIS
LIN {X 0.170,Y -488.959,Z 705.513,A 0.000,B 0.000,C 90.000,E1 272.236} C_DIS
LIN {X -0.113,Y -488.385,Z 705.510,A 0.000,B 0.000,C 90.000,E1 271.776} C_DIS
LIN {X 0.074,Y -487.414,Z 705.507,A 0.000,B 0.000,C 90.000,E1 271.260} C_DIS
LIN {X -0.229,Y -486.020,Z 705.504,A 0.000,B 0.000,C 90.000,E1 270.802} C_DIS
LIN {X -0.049,Y -484.241,Z 705.502,A 0.000,B 0.000,C 90.000,E1 270.286} C_DIS
LIN {X 0.121,Y -481.822,Z 705.499,A 0.000,B 0.000,C 90.000,E1 269.771} C_DIS
LIN {X -0.205,Y -478.812,Z 705.496,A 0.000,B 0.000,C 90.000,E1 269.312} C_DIS
LIN {X -0.067,Y -474.939,Z 705.493,A 0.000,B 0.000,C 90.000,E1 268.797} C_DIS
LIN {X 0.047,Y -470.106,Z 705.490,A 0.000,B 0.000,C 90.000,E1 268.282} C_DIS
LIN {X -0.068,Y -467.337,Z 705.489,A 0.000,B 0.000,C 90.000,E1 268.051} C_DIS
LIN {X -0.194,Y -464.196,Z 705.488,A 0.000,B 0.000,C 90.000,E1 267.822} C_DIS
LIN {X 0.102,Y -457.697,Z 705.485,A 0.000,B 0.000,C 90.000,E1 267.364} C_DIS
LIN {X 0.062,Y -454.469,Z 705.484,A 0.000,B 0.000,C 90.000,E1 267.192} C_DIS
LIN {X -0.172,Y -447.332,Z 705.483,A 0.000,B 0.000,C 90.000,E1 266.906} C_DIS
LIN {X 0.156,Y -439.924,Z 705.481,A 0.000,B 0.000,C 90.000,E1 266.617} C_DIS
LIN {X 0.032,Y -431.915,Z 705.480,A 0.000,B 0.000,C 90.000,E1 266.445} C_DIS
LIN {X -0.139,Y -426.586,Z 705.480,A 0.000,B 0.000,C 90.000,E1 266.388} C_DIS
LIN {X -0.201,Y -417.441,Z 705.479,A 0.000,B 0.000,C 90.000,E1 266.331} C_DIS
LIN {X 0.072,Y -180.935,Z 705.479,A 0.000,B 0.000,C 90.000,E1 266.274} C_DIS
LIN {X -0.081,Y -180.716,Z 705.470,A 0.000,B 0.000,C 90.000,E1 264.609} C_DIS
LIN {X 0.017,Y -178.804,Z 705.442,A 0.000,B 0.000,C 90.000,E1 259.511} C_DIS
LIN {X 0.093,Y -175.848,Z 705.413,A 0.000,B 0.000,C 90.000,E1 254.393} C_DIS
LIN {X 0.053,Y -172.584,Z 705.390,A 0.000,B 0.000,C 90.000,E1 250.134} C_DIS
LIN {X 0.069,Y -171.474,Z 705.380,A 0.000,B 0.000,C 90.000,E1 248.411} C_DIS
